LIN {X 0,Y 277.305,Z 271.444,A -85,B 0,C 180,E1 -17523.174,E2 -17523.174} C_VEL
LIN {X 0,Y 278.371,Z 274.382,A -85,B 0,C 180,E1 -17523.39,E2 -17523.39} C_VEL
LIN {X 0,Y 284.736,Z 287.887,A -85,B 0,C 180,E1 -17524.559,E2 -17524.559} C_VEL
LIN {X 0,Y 289.176,Z 296.03,A -85,B 0,C 180,E1 -17525.459,E2 -17525.459} C_VEL
LIN {X 0,Y 294.753,Z 304.53,A -85,B 0,C 180,E1 -17526.584,E2 -17526.584} C_VEL
LIN {X 0,Y 302.885,Z 314.906,A -85,B 0,C 180,E1 -17528.207,E2 -17528.207} C_VEL
LIN {X 0,Y 312.071,Z 325.664,A -85,B 0,C 180,E1 -17530.11,E2 -17530.11} C_VEL
LIN {X 0,Y 318.486,Z 332.585,A -85,B 0,C 180,E1 -17531.566,E2 -17531.566} C_VEL
LIN {X 0,Y 325.416,Z 339.712,A -85,B 0,C 180,E1 -17533.306,E2 -17533.306} C_VEL
LIN {X 0,Y 330.152,Z 344.132,A -85,B 0,C 180,E1 -17534.587,E2 -17534.587} C_VEL
LIN {X 0,Y 333.613,Z 347.56,A -85,B 0,C 180,E1 -17535.666,E2 -17535.666} C_VEL
LIN {X 0,Y 338.551,Z 351.983,A -85,B 0,C 180,E1 -17537.29,E2 -17537.29} C_VEL
LIN {X 0,Y 343.443,Z 356.189,A -85,B 0,C 180,E1 -17539.131,E2 -17539.131} C_VEL
LIN {X 0,Y 346.978,Z 358.993,A -85,B 0,C 180,E1 -17540.675,E2 -17540.675} C_VEL
LIN {X 0,Y 349.09,Z 361.115,A -85,B 0,C 180,E1 -17541.899,E2 -17541.899} C_VEL
LIN {X 0,Y 351.016,Z 362.827,A -85,B 0,C 180,E1 -17543.1,E2 -17543.1} C_VEL
LIN {X 0,Y 352.986,Z 364.25,A -85,B 0,C 180,E1 -17544.46,E2 -17544.46} C_VEL
LIN {X 0,Y 354.317,Z 364.994,A -85,B 0,C 180,E1 -17545.449,E2 -17545.449} C_VEL
LIN {X 0,Y 355.672,Z 365.56,A -85,B 0,C 180,E1 -17546.602,E2 -17546.602} C_VEL
LIN {X 0,Y 356.709,Z 365.873,A -85,B 0,C 180,E1 -17547.742,E2 -17547.742} C_VEL
LIN {X 0,Y 357.373,Z 366.011,A -85,B 0,C 180,E1 -17548.873,E2 -17548.873} C_VEL
LIN {X 0,Y 357.622,Z 366.036,A -85,B 0,C 180,E1 -17550,E2 -17550} C_VEL
LIN {X 0,Y 357.372,Z 366.013,A -85,B 0,C 180,E1 -17551.127,E2 -17551.127} C_VEL
LIN {X 0,Y 356.704,Z 365.874,A -85,B 0,C 180,E1 -17552.258,E2 -17552.258} C_VEL
LIN {X 0,Y 355.662,Z 365.563,A -85,B 0,C 180,E1 -17553.398,E2 -17553.398} C_VEL
LIN {X 0,Y 354.323,Z 364.997,A -85,B 0,C 180,E1 -17554.551,E2 -17554.551} C_VEL
LIN {X 0,Y 352.755,Z 364.109,A -85,B 0,C 180,E1 -17555.717,E2 -17555.717} C_VEL
LIN {X 0,Y 350.974,Z 362.834,A -85,B 0,C 180,E1 -17556.9,E2 -17556.9} C_VEL
LIN {X 0,Y 348.241,Z 360.258,A -85,B 0,C 180,E1 -17558.618,E2 -17558.618} C_VEL
LIN {X 0,Y 346.063,Z 358.167,A -85,B 0,C 180,E1 -17559.786,E2 -17559.786} C_VEL
LIN {X 0,Y 342.661,Z 355.63,A -85,B 0,C 180,E1 -17561.144,E2 -17561.144} C_VEL
LIN {X 0,Y 338.543,Z 351.93,A -85,B 0,C 180,E1 -17562.705,E2 -17562.705} C_VEL
LIN {X 0,Y 335.745,Z 349.331,A -85,B 0,C 180,E1 -17563.679,E2 -17563.679} C_VEL
LIN {X 0,Y 331.243,Z 345.273,A -85,B 0,C 180,E1 -17565.064,E2 -17565.064} C_VEL
LIN {X 0,Y 325.444,Z 339.675,A -85,B 0,C 180,E1 -17566.699,E2 -17566.699} C_VEL
LIN {X 0,Y 318.499,Z 332.541,A -85,B 0,C 180,E1 -17568.441,E2 -17568.441} C_VEL
LIN {X 0,Y 312.069,Z 325.652,A -85,B 0,C 180,E1 -17569.888,E2 -17569.888} C_VEL
LIN {X 0,Y 303.933,Z 316.233,A -85,B 0,C 180,E1 -17571.574,E2 -17571.574} C_VEL
LIN {X 0,Y 294.754,Z 304.541,A -85,B 0,C 180,E1 -17573.415,E2 -17573.415} C_VEL
LIN {X 0,Y 288.184,Z 294.427,A -85,B 0,C 180,E1 -17574.738,E2 -17574.738} C_VEL
LIN {X 0,Y 283.212,Z 284.587,A -85,B 0,C 180,E1 -17575.747,E2 -17575.747} C_VEL
LIN {X 0,Y 277.393,Z 272.078,A -85,B 0,C 180,E1 -17576.778,E2 -17576.778} C_VEL
LIN {X 0,Y 277.312,Z 271.443,A -85,B 0,C 180,E1 -17576.829,E2 -17576.829} C_VEL
LIN {X 0,Y 277.223,Z 271.454,A -85,B 0,C 180,E1 -17580.487,E2 -17580.487} C_VEL
LIN {X 0,Y 277.205,Z 271.457,A -85,B 0,C 180,E1 -17583.901,E2 -17583.901} C_VEL
LIN {X 0,Y 277.235,Z 271.451,A -85,B 0,C 180,E1 -17587.473,E2 -17587.473} C_VEL
LIN {X 0,Y 277.221,Z 271.451,A -85,B 0,C 180,E1 -17591.233,E2 -17591.233} C_VEL
LIN {X 0,Y 277.247,Z 271.448,A -85,B 0,C 180,E1 -17595.216,E2 -17595.216} C_VEL
LIN {X 0,Y 277.257,Z 271.449,A -85,B 0,C 180,E1 -17599.502,E2 -17599.502} C_VEL
LIN {X 0,Y 277.249,Z 271.448,A -85,B 0,C 180,E1 -17602.541,E2 -17602.541} C_VEL
LIN {X 0,Y 277.22,Z 271.451,A -85,B 0,C 180,E1 -17606.113,E2 -17606.113} C_VEL
LIN {X 0,Y 277.232,Z 271.453,A -85,B 0,C 180,E1 -17609.547,E2 -17609.547} C_VEL
LIN {X 0,Y 277.323,Z 271.439,A -85,B 0,C 180,E1 -17612.872,E2 -17612.872} C_VEL
LIN {X 0,Y 277.271,Z 271.444,A -85,B 0,C 180,E1 -17616.085,E2 -17616.085} C_VEL
LIN {X 0,Y 277.263,Z 271.443,A -85,B 0,C 180,E1 -17620.771,E2 -17620.771} C_VEL
LIN {X 0,Y 277.391,Z 271.43,A -85,B 0,C 180,E1 -17625.333,E2 -17625.333} C_VEL
LIN {X 0,Y 277.44,Z 271.421,A -85,B 0,C 180,E1 -17629.795,E2 -17629.795} C_VEL
LIN {X 0,Y 277.602,Z 271.406,A -85,B 0,C 180,E1 -17632.737,E2 -17632.737} C_VEL
LIN {X 0,Y 277.81,Z 271.365,A -85,B 0,C 180,E1 -17638.559,E2 -17638.559} C_VEL
LIN {X 0,Y 277.807,Z 271.377,A -85,B 0,C 180,E1 -17641.458,E2 -17641.458} C_VEL
LIN {X 0,Y 277.608,Z 271.404,A -85,B 0,C 180,E1 -17647.28,E2 -17647.28} C_VEL
LIN {X 0,Y 277.455,Z 271.425,A -85,B 0,C 180,E1 -17650.221,E2 -17650.221} C_VEL
LIN {X 0,Y 277.412,Z 271.431,A -85,B 0,C 180,E1 -17654.683,E2 -17654.683} C_VEL
LIN {X 0,Y 277.29,Z 271.443,A -85,B 0,C 180,E1 -17659.246,E2 -17659.246} C_VEL
LIN {X 0,Y 277.28,Z 271.448,A -85,B 0,C 180,E1 -17663.933,E2 -17663.933} C_VEL
LIN {X 0,Y 277.243,Z 271.447,A -85,B 0,C 180,E1 -17666.284,E2 -17666.284} C_VEL
LIN {X 0,Y 276.586,Z 271.534,A -85,B 0,C 180,E1 -17667.497,E2 -17667.497} C_VEL
LIN {X 0,Y 273.691,Z 271.893,A -85,B 0,C 180,E1 -17669.472,E2 -17669.472} C_VEL
LIN {X 0,Y 271.272,Z 272.333,A -85,B 0,C 180,E1 -17671.075,E2 -17671.075} C_VEL
LIN {X 0,Y 270.307,Z 272.789,A -85,B 0,C 180,E1 -17672.316,E2 -17672.316} C_VEL
LIN {X 0,Y 270.268,Z 272.974,A -85,B 0,C 180,E1 -17672.735,E2 -17672.735} C_VEL
LIN {X 0,Y 270.578,Z 275.102,A -85,B 0,C 180,E1 -17676.692,E2 -17676.692} C_VEL
LIN {X 0,Y 270.939,Z 277.348,A -85,B 0,C 180,E1 -17680.436,E2 -17680.436} C_VEL
LIN {X 0,Y 271.224,Z 279.969,A -85,B 0,C 180,E1 -17684.406,E2 -17684.406} C_VEL
LIN {X 0,Y 271.163,Z 282.305,A -85,B 0,C 180,E1 -17687.635,E2 -17687.635} C_VEL
LIN {X 0,Y 270.847,Z 285.048,A -85,B 0,C 180,E1 -17691.128,E2 -17691.128} C_VEL
LIN {X 0,Y 270.224,Z 288.327,A -85,B 0,C 180,E1 -17695.099,E2 -17695.099} C_VEL
LIN {X 0,Y 269.607,Z 292.063,A -85,B 0,C 180,E1 -17699.354,E2 -17699.354} C_VEL
LIN {X 0,Y 269.107,Z 295.022,A -85,B 0,C 180,E1 -17702.665,E2 -17702.665} C_VEL
LIN {X 0,Y 269.854,Z 298.046,A -85,B 0,C 180,E1 -17702.869,E2 -17702.869} C_VEL
LIN {X 0,Y 273.525,Z 311.599,A -85,B 0,C 180,E1 -17704.078,E2 -17704.078} C_VEL
LIN {X 0,Y 275.582,Z 321.927,A -85,B 0,C 180,E1 -17705.147,E2 -17705.147} C_VEL
LIN {X 0,Y 276.762,Z 330.171,A -85,B 0,C 180,E1 -17706.102,E2 -17706.102} C_VEL
LIN {X 0,Y 277.572,Z 339.948,A -85,B 0,C 180,E1 -17707.397,E2 -17707.397} C_VEL
LIN {X 0,Y 277.789,Z 344.628,A -85,B 0,C 180,E1 -17708.089,E2 -17708.089} C_VEL
LIN {X 0,Y 275.819,Z 355.141,A -85,B 0,C 180,E1 -17709.686,E2 -17709.686} C_VEL
LIN {X 0,Y 274.235,Z 363.639,A -85,B 0,C 180,E1 -17711.317,E2 -17711.317} C_VEL
LIN {X 0,Y 272.702,Z 371.465,A -85,B 0,C 180,E1 -17713.147,E2 -17713.147} C_VEL
LIN {X 0,Y 271.408,Z 378.004,A -85,B 0,C 180,E1 -17714.993,E2 -17714.993} C_VEL
LIN {X 0,Y 270.436,Z 382.504,A -85,B 0,C 180,E1 -17716.474,E2 -17716.474} C_VEL
LIN {X 0,Y 269.416,Z 387.997,A -85,B 0,C 180,E1 -17718.718,E2 -17718.718} C_VEL
LIN {X 0,Y 268.723,Z 392.325,A -85,B 0,C 180,E1 -17720.972,E2 -17720.972} C_VEL
LIN {X 0,Y 268.437,Z 394.694,A -85,B 0,C 180,E1 -17722.478,E2 -17722.478} C_VEL
LIN {X 0,Y 268.147,Z 397.425,A -85,B 0,C 180,E1 -17724.907,E2 -17724.907} C_VEL
LIN {X 0,Y 268.167,Z 398.948,A -85,B 0,C 180,E1 -17726.996,E2 -17726.996} C_VEL
LIN {X 0,Y 268.189,Z 399.539,A -85,B 0,C 180,E1 -17728.498,E2 -17728.498} C_VEL
LIN {X 0,Y 268.189,Z 399.539,A -85,B 0,C 180,E1 -17731.502,E2 -17731.502} C_VEL
LIN {X 0,Y 268.166,Z 398.948,A -85,B 0,C 180,E1 -17733.004,E2 -17733.004} C_VEL
LIN {X 0,Y 268.242,Z 396.496,A -85,B 0,C 180,E1 -17736.016,E2 -17736.016} C_VEL
LIN {X 0,Y 268.566,Z 393.543,A -85,B 0,C 180,E1 -17738.275,E2 -17738.275} C_VEL
LIN {X 0,Y 269.161,Z 389.552,A -85,B 0,C 180,E1 -17740.531,E2 -17740.531} C_VEL
LIN {X 0,Y 270.044,Z 384.42,A -85,B 0,C 180,E1 -17742.78,E2 -17742.78} C_VEL
LIN {X 0,Y 271.134,Z 379.159,A -85,B 0,C 180,E1 -17744.639,E2 -17744.639} C_VEL
LIN {X 0,Y 272.4,Z 372.841,A -85,B 0,C 180,E1 -17746.487,E2 -17746.487} C_VEL
LIN {X 0,Y 273.641,Z 366.891,A -85,B 0,C 180,E1 -17747.95,E2 -17747.95} C_VEL
LIN {X 0,Y 274.86,Z 359.961,A -85,B 0,C 180,E1 -17749.414,E2 -17749.414} C_VEL
LIN {X 0,Y 276.443,Z 351.784,A -85,B 0,C 180,E1 -17750.849,E2 -17750.849} C_VEL
LIN {X 0,Y 277.754,Z 344.627,A -85,B 0,C 180,E1 -17751.914,E2 -17751.914} C_VEL
LIN {X 0,Y 277.272,Z 335.68,A -85,B 0,C 180,E1 -17753.188,E2 -17753.188} C_VEL
LIN {X 0,Y 276.143,Z 325.328,A -85,B 0,C 180,E1 -17754.463,E2 -17754.463} C_VEL
LIN {X 0,Y 274.461,Z 315.993,A -85,B 0,C 180,E1 -17755.483,E2 -17755.483} C_VEL
LIN {X 0,Y 271.884,Z 305.118,A -85,B 0,C 180,E1 -17756.518,E2 -17756.518} C_VEL
LIN {X 0,Y 269.171,Z 295.65,A -85,B 0,C 180,E1 -17757.299,E2 -17757.299} C_VEL
LIN {X 0,Y 269.089,Z 295.013,A -85,B 0,C 180,E1 -17757.365,E2 -17757.365} C_VEL
LIN {X 0,Y 269.661,Z 291.299,A -85,B 0,C 180,E1 -17761.415,E2 -17761.415} C_VEL
LIN {X 0,Y 270.24,Z 288.287,A -85,B 0,C 180,E1 -17764.899,E2 -17764.899} C_VEL
LIN {X 0,Y 270.846,Z 285.017,A -85,B 0,C 180,E1 -17768.872,E2 -17768.872} C_VEL
LIN {X 0,Y 271.157,Z 282.304,A -85,B 0,C 180,E1 -17772.366,E2 -17772.366} C_VEL
LIN {X 0,Y 271.224,Z 279.957,A -85,B 0,C 180,E1 -17775.594,E2 -17775.594} C_VEL
LIN {X 0,Y 270.939,Z 277.339,A -85,B 0,C 180,E1 -17779.564,E2 -17779.564} C_VEL
LIN {X 0,Y 270.556,Z 274.906,A -85,B 0,C 180,E1 -17783.633,E2 -17783.633} C_VEL
LIN {X 0,Y 270.315,Z 273.144,A -85,B 0,C 180,E1 -17786.9,E2 -17786.9} C_VEL
LIN {X 0,Y 270.196,Z 272.332,A -85,B 0,C 180,E1 -17789.13,E2 -17789.13} C_VEL
LIN {X 0,Y 270.209,Z 272.329,A -85,B 0,C 180,E1 -17792.166,E2 -17792.166} C_VEL
LIN {X 0,Y 270.226,Z 272.327,A -85,B 0,C 180,E1 -17795.54,E2 -17795.54} C_VEL
LIN {X 0,Y 270.23,Z 272.325,A -85,B 0,C 180,E1 -17800.231,E2 -17800.231} C_VEL
LIN {X 0,Y 270.371,Z 272.305,A -85,B 0,C 180,E1 -17804.926,E2 -17804.926} C_VEL
LIN {X 0,Y 270.407,Z 272.304,A -85,B 0,C 180,E1 -17809.509,E2 -17809.509} C_VEL
LIN {X 0,Y 270.568,Z 272.28,A -85,B 0,C 180,E1 -17812.529,E2 -17812.529} C_VEL
LIN {X 0,Y 270.771,Z 272.253,A -85,B 0,C 180,E1 -17818.504,E2 -17818.504} C_VEL
LIN {X 0,Y 270.776,Z 272.239,A -85,B 0,C 180,E1 -17821.479,E2 -17821.479} C_VEL
LIN {X 0,Y 270.562,Z 272.282,A -85,B 0,C 180,E1 -17827.453,E2 -17827.453} C_VEL
LIN {X 0,Y 270.392,Z 272.3,A -85,B 0,C 180,E1 -17830.473,E2 -17830.473} C_VEL
LIN {X 0,Y 270.35,Z 272.307,A -85,B 0,C 180,E1 -17835.058,E2 -17835.058} C_VEL
LIN {X 0,Y 270.202,Z 272.321,A -85,B 0,C 180,E1 -17839.753,E2 -17839.753} C_VEL
LIN {X 0,Y 270.212,Z 272.324,A -85,B 0,C 180,E1 -17844.58,E2 -17844.58} C_VEL
LIN {X 0,Y 270.217,Z 272.324,A -85,B 0,C 180,E1 -17847.903,E2 -17847.903} C_VEL
LIN {X 0,Y 270.143,Z 272.333,A -85,B 0,C 180,E1 -17851.341,E2 -17851.341} C_VEL
LIN {X 0,Y 270.181,Z 272.329,A -85,B 0,C 180,E1 -17854.895,E2 -17854.895} C_VEL
LIN {X 0,Y 270.187,Z 272.329,A -85,B 0,C 180,E1 -17858.709,E2 -17858.709} C_VEL
LIN {X 0,Y 270.191,Z 272.329,A -85,B 0,C 180,E1 -17862.539,E2 -17862.539} C_VEL
LIN {X 0,Y 270.19,Z 272.327,A -85,B 0,C 180,E1 -17866.729,E2 -17866.729} C_VEL
LIN {X 0,Y 270.202,Z 272.326,A -85,B 0,C 180,E1 -17869.441,E2 -17869.441} C_VEL
LIN {X 0,Y 270.207,Z 272.328,A -85,B 0,C 180,E1 -17873.716,E2 -17873.716} C_VEL
LIN {X 0,Y 270.155,Z 272.333,A -85,B 0,C 180,E1 -17876.887,E2 -17876.887} C_VEL
LIN {X 0,Y 270.178,Z 272.331,A -85,B 0,C 180,E1 -17880.381,E2 -17880.381} C_VEL
LIN {X 0,Y 270.246,Z 272.322,A -85,B 0,C 180,E1 -17882.435,E2 -17882.435} C_VEL
LIN {X 0,Y 271.193,Z 275.036,A -85,B 0,C 180,E1 -17882.64,E2 -17882.64} C_VEL
LIN {X 0,Y 277.258,Z 287.788,A -85,B 0,C 180,E1 -17883.803,E2 -17883.803} C_VEL
LIN {X 0,Y 281.67,Z 296.983,A -85,B 0,C 180,E1 -17884.809,E2 -17884.809} C_VEL
LIN {X 0,Y 287.233,Z 305.985,A -85,B 0,C 180,E1 -17886.041,E2 -17886.041} C_VEL
LIN {X 0,Y 294.832,Z 316.369,A -85,B 0,C 180,E1 -17887.711,E2 -17887.711} C_VEL
LIN {X 0,Y 304.031,Z 327.199,A -85,B 0,C 180,E1 -17889.712,E2 -17889.712} C_VEL
LIN {X 0,Y 312.544,Z 336.483,A -85,B 0,C 180,E1 -17891.651,E2 -17891.651} C_VEL
LIN {X 0,Y 318.048,Z 342.107,A -85,B 0,C 180,E1 -17893.005,E2 -17893.005} C_VEL
LIN {X 0,Y 324.198,Z 348.021,A -85,B 0,C 180,E1 -17894.649,E2 -17894.649} C_VEL
LIN {X 0,Y 328.692,Z 352.374,A -85,B 0,C 180,E1 -17896.035,E2 -17896.035} C_VEL
LIN {X 0,Y 333.966,Z 357.233,A -85,B 0,C 180,E1 -17897.852,E2 -17897.852} C_VEL
LIN {X 0,Y 338.688,Z 361.032,A -85,B 0,C 180,E1 -17899.64,E2 -17899.64} C_VEL
LIN {X 0,Y 341.529,Z 363.397,A -85,B 0,C 180,E1 -17900.955,E2 -17900.955} C_VEL
LIN {X 0,Y 344.893,Z 366.614,A -85,B 0,C 180,E1 -17902.977,E2 -17902.977} C_VEL
LIN {X 0,Y 346.673,Z 368.004,A -85,B 0,C 180,E1 -17904.182,E2 -17904.182} C_VEL
LIN {X 0,Y 348.314,Z 368.949,A -85,B 0,C 180,E1 -17905.371,E2 -17905.371} C_VEL
LIN {X 0,Y 349.715,Z 369.542,A -85,B 0,C 180,E1 -17906.544,E2 -17906.544} C_VEL
LIN {X 0,Y 350.797,Z 369.895,A -85,B 0,C 180,E1 -17907.704,E2 -17907.704} C_VEL
LIN {X 0,Y 351.516,Z 370.064,A -85,B 0,C 180,E1 -17908.854,E2 -17908.854} C_VEL
LIN {X 0,Y 351.802,Z 370.093,A -85,B 0,C 180,E1 -17910,E2 -17910} C_VEL
LIN {X 0,Y 351.428,Z 370.042,A -85,B 0,C 180,E1 -17911.304,E2 -17911.304} C_VEL
LIN {X 0,Y 350.795,Z 369.894,A -85,B 0,C 180,E1 -17912.296,E2 -17912.296} C_VEL
LIN {X 0,Y 349.687,Z 369.557,A -85,B 0,C 180,E1 -17913.457,E2 -17913.457} C_VEL
LIN {X 0,Y 348.32,Z 368.954,A -85,B 0,C 180,E1 -17914.629,E2 -17914.629} C_VEL
LIN {X 0,Y 346.271,Z 367.704,A -85,B 0,C 180,E1 -17916.102,E2 -17916.102} C_VEL
LIN {X 0,Y 342.923,Z 364.794,A -85,B 0,C 180,E1 -17918.248,E2 -17918.248} C_VEL
LIN {X 0,Y 340.682,Z 362.566,A -85,B 0,C 180,E1 -17919.499,E2 -17919.499} C_VEL
LIN {X 0,Y 336.609,Z 359.463,A -85,B 0,C 180,E1 -17921.151,E2 -17921.151} C_VEL
LIN {X 0,Y 333.301,Z 356.536,A -85,B 0,C 180,E1 -17922.404,E2 -17922.404} C_VEL
LIN {X 0,Y 328.614,Z 352.291,A -85,B 0,C 180,E1 -17923.982,E2 -17923.982} C_VEL
LIN {X 0,Y 323.151,Z 347.015,A -85,B 0,C 180,E1 -17925.649,E2 -17925.649} C_VEL
LIN {X 0,Y 316.588,Z 340.622,A -85,B 0,C 180,E1 -17927.374,E2 -17927.374} C_VEL
LIN {X 0,Y 310.388,Z 334.142,A -85,B 0,C 180,E1 -17928.866,E2 -17928.866} C_VEL
LIN {X 0,Y 300.983,Z 323.659,A -85,B 0,C 180,E1 -17930.963,E2 -17930.963} C_VEL
LIN {X 0,Y 292.248,Z 312.969,A -85,B 0,C 180,E1 -17932.863,E2 -17932.863} C_VEL
LIN {X 0,Y 285.391,Z 303.244,A -85,B 0,C 180,E1 -17934.362,E2 -17934.362} C_VEL
LIN {X 0,Y 279.96,Z 293.672,A -85,B 0,C 180,E1 -17935.584,E2 -17935.584} C_VEL
LIN {X 0,Y 273.934,Z 280.583,A -85,B 0,C 180,E1 -17936.873,E2 -17936.873} C_VEL
LIN {X 0,Y 270.418,Z 273.239,A -85,B 0,C 180,E1 -17937.498,E2 -17937.498} C_VEL
LIN {X 0,Y 270.232,Z 272.324,A -85,B 0,C 180,E1 -17937.598,E2 -17937.598} C_VEL
LIN {X 0,Y 270.135,Z 272.335,A -85,B 0,C 180,E1 -17941.354,E2 -17941.354} C_VEL
LIN {X 0,Y 270.166,Z 272.331,A -85,B 0,C 180,E1 -17944.91,E2 -17944.91} C_VEL
LIN {X 0,Y 270.178,Z 272.329,A -85,B 0,C 180,E1 -17948.723,E2 -17948.723} C_VEL
LIN {X 0,Y 270.187,Z 272.328,A -85,B 0,C 180,E1 -17952.554,E2 -17952.554} C_VEL
LIN {X 0,Y 270.192,Z 272.327,A -85,B 0,C 180,E1 -17956.743,E2 -17956.743} C_VEL
LIN {X 0,Y 270.209,Z 272.327,A -85,B 0,C 180,E1 -17959.455,E2 -17959.455} C_VEL
LIN {X 0,Y 270.221,Z 272.326,A -85,B 0,C 180,E1 -17963.73,E2 -17963.73} C_VEL
LIN {X 0,Y 270.17,Z 272.329,A -85,B 0,C 180,E1 -17966.901,E2 -17966.901} C_VEL
LIN {X 0,Y 270.162,Z 272.331,A -85,B 0,C 180,E1 -17970.391,E2 -17970.391} C_VEL
LIN {X 0,Y 270.229,Z 272.322,A -85,B 0,C 180,E1 -17973.772,E2 -17973.772} C_VEL
LIN {X 0,Y 270.182,Z 272.329,A -85,B 0,C 180,E1 -17977.045,E2 -17977.045} C_VEL
LIN {X 0,Y 270.202,Z 272.321,A -85,B 0,C 180,E1 -17980.247,E2 -17980.247} C_VEL
LIN {X 0,Y 270.35,Z 272.307,A -85,B 0,C 180,E1 -17984.942,E2 -17984.942} C_VEL
LIN {X 0,Y 270.392,Z 272.3,A -85,B 0,C 180,E1 -17989.527,E2 -17989.527} C_VEL
LIN {X 0,Y 270.562,Z 272.282,A -85,B 0,C 180,E1 -17992.547,E2 -17992.547} C_VEL
LIN {X 0,Y 270.776,Z 272.239,A -85,B 0,C 180,E1 -17998.521,E2 -17998.521} C_VEL
LIN {X 0,Y 270.771,Z 272.253,A -85,B 0,C 180,E1 -18001.496,E2 -18001.496} C_VEL
LIN {X 0,Y 270.568,Z 272.28,A -85,B 0,C 180,E1 -18007.471,E2 -18007.471} C_VEL
LIN {X 0,Y 270.407,Z 272.305,A -85,B 0,C 180,E1 -18010.491,E2 -18010.491} C_VEL
LIN {X 0,Y 270.371,Z 272.306,A -85,B 0,C 180,E1 -18015.074,E2 -18015.074} C_VEL
LIN {X 0,Y 270.229,Z 272.324,A -85,B 0,C 180,E1 -18019.769,E2 -18019.769} C_VEL
LIN {X 0,Y 270.207,Z 272.328,A -85,B 0,C 180,E1 -18024.6,E2 -18024.6} C_VEL
LIN {X 0,Y 270.206,Z 272.328,A -85,B 0,C 180,E1 -18027.924,E2 -18027.924} C_VEL
LIN {X 0,Y 270.187,Z 272.334,A -85,B 0,C 180,E1 -18031.356,E2 -18031.356} C_VEL
LIN {X 0,Y 270.268,Z 272.974,A -85,B 0,C 180,E1 -18032.735,E2 -18032.735} C_VEL
LIN {X 0,Y 269.724,Z 273.708,A -85,B 0,C 180,E1 -18033.973,E2 -18033.973} C_VEL
LIN {X 0,Y 267.004,Z 275.236,A -85,B 0,C 180,E1 -18035.983,E2 -18035.983} C_VEL
LIN {X 0,Y 264.697,Z 276.523,A -85,B 0,C 180,E1 -18037.616,E2 -18037.616} C_VEL
LIN {X 0,Y 263.792,Z 277.402,A -85,B 0,C 180,E1 -18038.882,E2 -18038.882} C_VEL
LIN {X 0,Y 263.768,Z 277.665,A -85,B 0,C 180,E1 -18039.311,E2 -18039.311} C_VEL
LIN {X 0,Y 263.995,Z 279.198,A -85,B 0,C 180,E1 -18041.807,E2 -18041.807} C_VEL
LIN {X 0,Y 264.161,Z 280.692,A -85,B 0,C 180,E1 -18044.084,E2 -18044.084} C_VEL
LIN {X 0,Y 264.182,Z 282.173,A -85,B 0,C 180,E1 -18046.239,E2 -18046.239} C_VEL
LIN {X 0,Y 264.084,Z 283.666,A -85,B 0,C 180,E1 -18048.294,E2 -18048.294} C_VEL
LIN {X 0,Y 263.6,Z 286.669,A -85,B 0,C 180,E1 -18052.179,E2 -18052.179} C_VEL
LIN {X 0,Y 263.009,Z 289.753,A -85,B 0,C 180,E1 -18055.942,E2 -18055.942} C_VEL
LIN {X 0,Y 262.512,Z 292.712,A -85,B 0,C 180,E1 -18059.426,E2 -18059.426} C_VEL
LIN {X 0,Y 262.102,Z 294.933,A -85,B 0,C 180,E1 -18061.88,E2 -18061.88} C_VEL
LIN {X 0,Y 263.003,Z 298.178,A -85,B 0,C 180,E1 -18062.116,E2 -18062.116} C_VEL
LIN {X 0,Y 266.675,Z 311.678,A -85,B 0,C 180,E1 -18063.384,E2 -18063.384} C_VEL
LIN {X 0,Y 268.682,Z 321.718,A -85,B 0,C 180,E1 -18064.464,E2 -18064.464} C_VEL
LIN {X 0,Y 270.078,Z 331.206,A -85,B 0,C 180,E1 -18065.626,E2 -18065.626} C_VEL
LIN {X 0,Y 270.79,Z 339.979,A -85,B 0,C 180,E1 -18066.833,E2 -18066.833} C_VEL
LIN {X 0,Y 270.977,Z 345.785,A -85,B 0,C 180,E1 -18067.71,E2 -18067.71} C_VEL
LIN {X 0,Y 268.939,Z 355.928,A -85,B 0,C 180,E1 -18069.343,E2 -18069.343} C_VEL
LIN {X 0,Y 267.111,Z 365.231,A -85,B 0,C 180,E1 -18071.238,E2 -18071.238} C_VEL
LIN {X 0,Y 265.889,Z 371.318,A -85,B 0,C 180,E1 -18072.715,E2 -18072.715} C_VEL
LIN {X 0,Y 264.53,Z 377.808,A -85,B 0,C 180,E1 -18074.593,E2 -18074.593} C_VEL
LIN {X 0,Y 263.527,Z 382.309,A -85,B 0,C 180,E1 -18076.113,E2 -18076.113} C_VEL
LIN {X 0,Y 262.425,Z 387.802,A -85,B 0,C 180,E1 -18078.413,E2 -18078.413} C_VEL
LIN {X 0,Y 261.702,Z 392.13,A -85,B 0,C 180,E1 -18080.728,E2 -18080.728} C_VEL
LIN {X 0,Y 261.372,Z 394.499,A -85,B 0,C 180,E1 -18082.274,E2 -18082.274} C_VEL
LIN {X 0,Y 261.046,Z 397.423,A -85,B 0,C 180,E1 -18085.02,E2 -18085.02} C_VEL
LIN {X 0,Y 261.062,Z 398.753,A -85,B 0,C 180,E1 -18086.914,E2 -18086.914} C_VEL
LIN {X 0,Y 261.095,Z 399.345,A -85,B 0,C 180,E1 -18088.458,E2 -18088.458} C_VEL
LIN {X 0,Y 261.095,Z 399.345,A -85,B 0,C 180,E1 -18091.542,E2 -18091.542} C_VEL
LIN {X 0,Y 261.061,Z 398.753,A -85,B 0,C 180,E1 -18093.086,E2 -18093.086} C_VEL
LIN {X 0,Y 261.17,Z 396.301,A -85,B 0,C 180,E1 -18096.179,E2 -18096.179} C_VEL
LIN {X 0,Y 261.528,Z 393.348,A -85,B 0,C 180,E1 -18098.499,E2 -18098.499} C_VEL
LIN {X 0,Y 262.137,Z 389.356,A -85,B 0,C 180,E1 -18100.817,E2 -18100.817} C_VEL
LIN {X 0,Y 263.103,Z 384.224,A -85,B 0,C 180,E1 -18103.123,E2 -18103.123} C_VEL
LIN {X 0,Y 264.253,Z 378.963,A -85,B 0,C 180,E1 -18105.029,E2 -18105.029} C_VEL
LIN {X 0,Y 265.586,Z 372.646,A -85,B 0,C 180,E1 -18106.922,E2 -18106.922} C_VEL
LIN {X 0,Y 266.839,Z 366.695,A -85,B 0,C 180,E1 -18108.424,E2 -18108.424} C_VEL
LIN {X 0,Y 268.137,Z 359.766,A -85,B 0,C 180,E1 -18109.921,E2 -18109.921} C_VEL
LIN {X 0,Y 269.814,Z 351.589,A -85,B 0,C 180,E1 -18111.386,E2 -18111.386} C_VEL
LIN {X 0,Y 270.986,Z 344.427,A -85,B 0,C 180,E1 -18112.49,E2 -18112.49} C_VEL
LIN {X 0,Y 270.41,Z 335.182,A -85,B 0,C 180,E1 -18113.849,E2 -18113.849} C_VEL
LIN {X 0,Y 269.366,Z 325.614,A -85,B 0,C 180,E1 -18115.071,E2 -18115.071} C_VEL
LIN {X 0,Y 267.439,Z 315.176,A -85,B 0,C 180,E1 -18116.252,E2 -18116.252} C_VEL
LIN {X 0,Y 265.009,Z 305.206,A -85,B 0,C 180,E1 -18117.244,E2 -18117.244} C_VEL
LIN {X 0,Y 262.166,Z 295.677,A -85,B 0,C 180,E1 -18118.082,E2 -18118.082} C_VEL
LIN {X 0,Y 262.101,Z 294.855,A -85,B 0,C 180,E1 -18118.14,E2 -18118.14} C_VEL
LIN {X 0,Y 262.547,Z 292.237,A -85,B 0,C 180,E1 -18121.052,E2 -18121.052} C_VEL
LIN {X 0,Y 263.02,Z 289.659,A -85,B 0,C 180,E1 -18124.133,E2 -18124.133} C_VEL
LIN {X 0,Y 263.6,Z 286.643,A -85,B 0,C 180,E1 -18127.821,E2 -18127.821} C_VEL
LIN {X 0,Y 264.084,Z 283.661,A -85,B 0,C 180,E1 -18131.706,E2 -18131.706} C_VEL
LIN {X 0,Y 264.186,Z 281.942,A -85,B 0,C 180,E1 -18134.079,E2 -18134.079} C_VEL
LIN {X 0,Y 264.144,Z 280.466,A -85,B 0,C 180,E1 -18136.22,E2 -18136.22} C_VEL
LIN {X 0,Y 264.015,Z 279.143,A -85,B 0,C 180,E1 -18138.271,E2 -18138.271} C_VEL
LIN {X 0,Y 263.644,Z 276.792,A -85,B 0,C 180,E1 -18142.176,E2 -18142.176} C_VEL
LIN {X 0,Y 263.361,Z 274.743,A -85,B 0,C 180,E1 -18145.908,E2 -18145.908} C_VEL
LIN {X 0,Y 263.161,Z 273.351,A -85,B 0,C 180,E1 -18148.713,E2 -18148.713} C_VEL
LIN {X 0,Y 263.137,Z 273.207,A -85,B 0,C 180,E1 -18152.988,E2 -18152.988} C_VEL
LIN {X 0,Y 263.145,Z 273.208,A -85,B 0,C 180,E1 -18156.375,E2 -18156.375} C_VEL
LIN {X 0,Y 263.215,Z 273.201,A -85,B 0,C 180,E1 -18159.681,E2 -18159.681} C_VEL
LIN {X 0,Y 263.314,Z 273.184,A -85,B 0,C 180,E1 -18164.511,E2 -18164.511} C_VEL
LIN {X 0,Y 263.346,Z 273.182,A -85,B 0,C 180,E1 -18169.225,E2 -18169.225} C_VEL
LIN {X 0,Y 263.531,Z 273.157,A -85,B 0,C 180,E1 -18172.329,E2 -18172.329} C_VEL
LIN {X 0,Y 263.734,Z 273.129,A -85,B 0,C 180,E1 -18178.464,E2 -18178.464} C_VEL
LIN {X 0,Y 263.74,Z 273.114,A -85,B 0,C 180,E1 -18181.518,E2 -18181.518} C_VEL
LIN {X 0,Y 263.523,Z 273.158,A -85,B 0,C 180,E1 -18187.654,E2 -18187.654} C_VEL
LIN {X 0,Y 263.331,Z 273.181,A -85,B 0,C 180,E1 -18190.758,E2 -18190.758} C_VEL
LIN {X 0,Y 263.292,Z 273.186,A -85,B 0,C 180,E1 -18195.471,E2 -18195.471} C_VEL
LIN {X 0,Y 263.187,Z 273.196,A -85,B 0,C 180,E1 -18200.302,E2 -18200.302} C_VEL
LIN {X 0,Y 263.165,Z 273.2,A -85,B 0,C 180,E1 -18205.284,E2 -18205.284} C_VEL
LIN {X 0,Y 263.126,Z 273.21,A -85,B 0,C 180,E1 -18208.724,E2 -18208.724} C_VEL
LIN {X 0,Y 263.097,Z 273.214,A -85,B 0,C 180,E1 -18212.28,E2 -18212.28} C_VEL
LIN {X 0,Y 263.154,Z 273.205,A -85,B 0,C 180,E1 -18215.97,E2 -18215.97} C_VEL
LIN {X 0,Y 263.123,Z 273.21,A -85,B 0,C 180,E1 -18219.855,E2 -18219.855} C_VEL
LIN {X 0,Y 263.151,Z 273.207,A -85,B 0,C 180,E1 -18223.962,E2 -18223.962} C_VEL
LIN {X 0,Y 263.128,Z 273.211,A -85,B 0,C 180,E1 -18228.109,E2 -18228.109} C_VEL
LIN {X 0,Y 263.142,Z 273.209,A -85,B 0,C 180,E1 -18232.101,E2 -18232.101} C_VEL
LIN {X 0,Y 263.137,Z 273.209,A -85,B 0,C 180,E1 -18235.884,E2 -18235.884} C_VEL
LIN {X 0,Y 263.101,Z 273.213,A -85,B 0,C 180,E1 -18239.501,E2 -18239.501} C_VEL
LIN {X 0,Y 263.174,Z 273.347,A -85,B 0,C 180,E1 -18241.674,E2 -18241.674} C_VEL
LIN {X 0,Y 264.168,Z 276.039,A -85,B 0,C 180,E1 -18241.873,E2 -18241.873} C_VEL
LIN {X 0,Y 270.002,Z 287.895,A -85,B 0,C 180,E1 -18243.037,E2 -18243.037} C_VEL
LIN {X 0,Y 274.745,Z 298.532,A -85,B 0,C 180,E1 -18244.224,E2 -18244.224} C_VEL
LIN {X 0,Y 279.966,Z 307.797,A -85,B 0,C 180,E1 -18245.523,E2 -18245.523} C_VEL
LIN {X 0,Y 286.211,Z 316.753,A -85,B 0,C 180,E1 -18247.016,E2 -18247.016} C_VEL
LIN {X 0,Y 294.917,Z 327.456,A -85,B 0,C 180,E1 -18249.056,E2 -18249.056} C_VEL
LIN {X 0,Y 304.221,Z 337.698,A -85,B 0,C 180,E1 -18251.257,E2 -18251.257} C_VEL
LIN {X 0,Y 311.996,Z 345.716,A -85,B 0,C 180,E1 -18253.166,E2 -18253.166} C_VEL
LIN {X 0,Y 318.525,Z 352.006,A -85,B 0,C 180,E1 -18254.938,E2 -18254.938} C_VEL
LIN {X 0,Y 322.402,Z 355.804,A -85,B 0,C 180,E1 -18256.126,E2 -18256.126} C_VEL
LIN {X 0,Y 326.785,Z 359.743,A -85,B 0,C 180,E1 -18257.581,E2 -18257.581} C_VEL
LIN {X 0,Y 330.501,Z 363.053,A -85,B 0,C 180,E1 -18258.967,E2 -18258.967} C_VEL
LIN {X 0,Y 334.685,Z 366.228,A -85,B 0,C 180,E1 -18260.666,E2 -18260.666} C_VEL
LIN {X 0,Y 338.411,Z 369.858,A -85,B 0,C 180,E1 -18262.842,E2 -18262.842} C_VEL
LIN {X 0,Y 340.265,Z 371.35,A -85,B 0,C 180,E1 -18264.073,E2 -18264.073} C_VEL
LIN {X 0,Y 341.945,Z 372.35,A -85,B 0,C 180,E1 -18265.284,E2 -18265.284} C_VEL
LIN {X 0,Y 343.406,Z 373.025,A -85,B 0,C 180,E1 -18266.48,E2 -18266.48} C_VEL
LIN {X 0,Y 344.592,Z 373.444,A -85,B 0,C 180,E1 -18267.679,E2 -18267.679} C_VEL
LIN {X 0,Y 345.365,Z 373.648,A -85,B 0,C 180,E1 -18268.834,E2 -18268.834} C_VEL
LIN {X 0,Y 345.687,Z 373.691,A -85,B 0,C 180,E1 -18270,E2 -18270} C_VEL
LIN {X 0,Y 345.385,Z 373.638,A -85,B 0,C 180,E1 -18271.166,E2 -18271.166} C_VEL
LIN {X 0,Y 344.56,Z 373.447,A -85,B 0,C 180,E1 -18272.338,E2 -18272.338} C_VEL
LIN {X 0,Y 343.372,Z 373.043,A -85,B 0,C 180,E1 -18273.52,E2 -18273.52} C_VEL
LIN {X 0,Y 341.954,Z 372.356,A -85,B 0,C 180,E1 -18274.715,E2 -18274.715} C_VEL
LIN {X 0,Y 339.444,Z 370.751,A -85,B 0,C 180,E1 -18276.47,E2 -18276.47} C_VEL
LIN {X 0,Y 336.389,Z 367.91,A -85,B 0,C 180,E1 -18278.409,E2 -18278.409} C_VEL
LIN {X 0,Y 333.836,Z 365.618,A -85,B 0,C 180,E1 -18279.696,E2 -18279.696} C_VEL
LIN {X 0,Y 328.688,Z 361.483,A -85,B 0,C 180,E1 -18281.719,E2 -18281.719} C_VEL
LIN {X 0,Y 323.601,Z 356.804,A -85,B 0,C 180,E1 -18283.51,E2 -18283.51} C_VEL
LIN {X 0,Y 318.506,Z 352.015,A -85,B 0,C 180,E1 -18285.07,E2 -18285.07} C_VEL
LIN {X 0,Y 311.999,Z 345.711,A -85,B 0,C 180,E1 -18286.836,E2 -18286.836} C_VEL
LIN {X 0,Y 303.534,Z 336.933,A -85,B 0,C 180,E1 -18288.914,E2 -18288.914} C_VEL
LIN {X 0,Y 292.987,Z 325.208,A -85,B 0,C 180,E1 -18291.392,E2 -18291.392} C_VEL
LIN {X 0,Y 284.418,Z 314.381,A -85,B 0,C 180,E1 -18293.408,E2 -18293.408} C_VEL
LIN {X 0,Y 278.042,Z 304.538,A -85,B 0,C 180,E1 -18294.961,E2 -18294.961} C_VEL
LIN {X 0,Y 273.081,Z 295.141,A -85,B 0,C 180,E1 -18296.19,E2 -18296.19} C_VEL
LIN {X 0,Y 267.373,Z 282.256,A -85,B 0,C 180,E1 -18297.529,E2 -18297.529} C_VEL
LIN {X 0,Y 263.315,Z 274.054,A -85,B 0,C 180,E1 -18298.288,E2 -18298.288} C_VEL
LIN {X 0,Y 263.15,Z 273.208,A -85,B 0,C 180,E1 -18298.367,E2 -18298.367} C_VEL
LIN {X 0,Y 263.084,Z 273.216,A -85,B 0,C 180,E1 -18302.294,E2 -18302.294} C_VEL
LIN {X 0,Y 263.14,Z 273.209,A -85,B 0,C 180,E1 -18305.985,E2 -18305.985} C_VEL
LIN {X 0,Y 263.117,Z 273.212,A -85,B 0,C 180,E1 -18309.869,E2 -18309.869} C_VEL
LIN {X 0,Y 263.15,Z 273.207,A -85,B 0,C 180,E1 -18313.977,E2 -18313.977} C_VEL
LIN {X 0,Y 263.133,Z 273.209,A -85,B 0,C 180,E1 -18318.124,E2 -18318.124} C_VEL
LIN {X 0,Y 263.153,Z 273.206,A -85,B 0,C 180,E1 -18322.116,E2 -18322.116} C_VEL
LIN {X 0,Y 263.152,Z 273.205,A -85,B 0,C 180,E1 -18325.899,E2 -18325.899} C_VEL
LIN {X 0,Y 263.098,Z 273.213,A -85,B 0,C 180,E1 -18329.513,E2 -18329.513} C_VEL
LIN {X 0,Y 263.161,Z 273.204,A -85,B 0,C 180,E1 -18333.011,E2 -18333.011} C_VEL
LIN {X 0,Y 263.128,Z 273.206,A -85,B 0,C 180,E1 -18336.393,E2 -18336.393} C_VEL
LIN {X 0,Y 263.187,Z 273.196,A -85,B 0,C 180,E1 -18339.698,E2 -18339.698} C_VEL
LIN {X 0,Y 263.292,Z 273.186,A -85,B 0,C 180,E1 -18344.529,E2 -18344.529} C_VEL
LIN {X 0,Y 263.331,Z 273.181,A -85,B 0,C 180,E1 -18349.242,E2 -18349.242} C_VEL
LIN {X 0,Y 263.523,Z 273.158,A -85,B 0,C 180,E1 -18352.346,E2 -18352.346} C_VEL
LIN {X 0,Y 263.74,Z 273.114,A -85,B 0,C 180,E1 -18358.482,E2 -18358.482} C_VEL
LIN {X 0,Y 263.734,Z 273.129,A -85,B 0,C 180,E1 -18361.536,E2 -18361.536} C_VEL
LIN {X 0,Y 263.531,Z 273.157,A -85,B 0,C 180,E1 -18367.671,E2 -18367.671} C_VEL
LIN {X 0,Y 263.346,Z 273.183,A -85,B 0,C 180,E1 -18370.775,E2 -18370.775} C_VEL
LIN {X 0,Y 263.314,Z 273.185,A -85,B 0,C 180,E1 -18375.489,E2 -18375.489} C_VEL
LIN {X 0,Y 263.215,Z 273.2,A -85,B 0,C 180,E1 -18380.319,E2 -18380.319} C_VEL
LIN {X 0,Y 263.145,Z 273.208,A -85,B 0,C 180,E1 -18385.306,E2 -18385.306} C_VEL
LIN {X 0,Y 263.14,Z 273.208,A -85,B 0,C 180,E1 -18388.743,E2 -18388.743} C_VEL
LIN {X 0,Y 263.161,Z 273.35,A -85,B 0,C 180,E1 -18391.287,E2 -18391.287} C_VEL
LIN {X 0,Y 263.359,Z 274.803,A -85,B 0,C 180,E1 -18394.183,E2 -18394.183} C_VEL
LIN {X 0,Y 263.644,Z 276.792,A -85,B 0,C 180,E1 -18397.824,E2 -18397.824} C_VEL
LIN {X 0,Y 263.768,Z 277.665,A -85,B 0,C 180,E1 -18399.311,E2 -18399.311} C_VEL
LIN {X 0,Y 263.263,Z 278.518,A -85,B 0,C 180,E1 -18400.574,E2 -18400.574} C_VEL
LIN {X 0,Y 260.575,Z 280.205,A -85,B 0,C 180,E1 -18402.627,E2 -18402.627} C_VEL
LIN {X 0,Y 258.203,Z 281.62,A -85,B 0,C 180,E1 -18404.295,E2 -18404.295} C_VEL
LIN {X 0,Y 257.168,Z 282.625,A -85,B 0,C 180,E1 -18405.588,E2 -18405.588} C_VEL
LIN {X 0,Y 257.08,Z 282.933,A -85,B 0,C 180,E1 -18406.027,E2 -18406.027} C_VEL
LIN {X 0,Y 256.933,Z 285.015,A -85,B 0,C 180,E1 -18408.969,E2 -18408.969} C_VEL
LIN {X 0,Y 256.442,Z 288.006,A -85,B 0,C 180,E1 -18412.921,E2 -18412.921} C_VEL
LIN {X 0,Y 255.797,Z 291.034,A -85,B 0,C 180,E1 -18416.668,E2 -18416.668} C_VEL
LIN {X 0,Y 255.237,Z 294.013,A -85,B 0,C 180,E1 -18420.289,E2 -18420.289} C_VEL
LIN {X 0,Y 255.11,Z 294.669,A -85,B 0,C 180,E1 -18421.035,E2 -18421.035} C_VEL
LIN {X 0,Y 255.933,Z 297.831,A -85,B 0,C 180,E1 -18421.27,E2 -18421.27} C_VEL
LIN {X 0,Y 259.545,Z 310.443,A -85,B 0,C 180,E1 -18422.507,E2 -18422.507} C_VEL
LIN {X 0,Y 261.851,Z 321.51,A -85,B 0,C 180,E1 -18423.747,E2 -18423.747} C_VEL
LIN {X 0,Y 263.228,Z 330.757,A -85,B 0,C 180,E1 -18424.917,E2 -18424.917} C_VEL
LIN {X 0,Y 264.015,Z 339.999,A -85,B 0,C 180,E1 -18426.236,E2 -18426.236} C_VEL
LIN {X 0,Y 264.199,Z 346.851,A -85,B 0,C 180,E1 -18427.312,E2 -18427.312} C_VEL
LIN {X 0,Y 262.31,Z 355.733,A -85,B 0,C 180,E1 -18428.796,E2 -18428.796} C_VEL
LIN {X 0,Y 260.393,Z 364.871,A -85,B 0,C 180,E1 -18430.694,E2 -18430.694} C_VEL
LIN {X 0,Y 258.775,Z 372.451,A -85,B 0,C 180,E1 -18432.618,E2 -18432.618} C_VEL
LIN {X 0,Y 257.385,Z 378.768,A -85,B 0,C 180,E1 -18434.56,E2 -18434.56} C_VEL
LIN {X 0,Y 256.151,Z 384.029,A -85,B 0,C 180,E1 -18436.514,E2 -18436.514} C_VEL
LIN {X 0,Y 255.132,Z 389.161,A -85,B 0,C 180,E1 -18438.883,E2 -18438.883} C_VEL
LIN {X 0,Y 254.485,Z 393.153,A -85,B 0,C 180,E1 -18441.264,E2 -18441.264} C_VEL
LIN {X 0,Y 254.085,Z 396.105,A -85,B 0,C 180,E1 -18443.648,E2 -18443.648} C_VEL
LIN {X 0,Y 253.96,Z 398.558,A -85,B 0,C 180,E1 -18446.827,E2 -18446.827} C_VEL
LIN {X 0,Y 254.003,Z 399.15,A -85,B 0,C 180,E1 -18448.415,E2 -18448.415} C_VEL
LIN {X 0,Y 254.043,Z 399.306,A -85,B 0,C 180,E1 -18450,E2 -18450} C_VEL
LIN {X 0,Y 254.003,Z 399.15,A -85,B 0,C 180,E1 -18451.585,E2 -18451.585} C_VEL
LIN {X 0,Y 253.959,Z 398.558,A -85,B 0,C 180,E1 -18453.173,E2 -18453.173} C_VEL
LIN {X 0,Y 254.082,Z 396.105,A -85,B 0,C 180,E1 -18456.352,E2 -18456.352} C_VEL
LIN {X 0,Y 254.485,Z 393.153,A -85,B 0,C 180,E1 -18458.736,E2 -18458.736} C_VEL
LIN {X 0,Y 255.132,Z 389.161,A -85,B 0,C 180,E1 -18461.117,E2 -18461.117} C_VEL
LIN {X 0,Y 256.151,Z 384.029,A -85,B 0,C 180,E1 -18463.486,E2 -18463.486} C_VEL
LIN {X 0,Y 257.384,Z 378.768,A -85,B 0,C 180,E1 -18465.44,E2 -18465.44} C_VEL
LIN {X 0,Y 258.794,Z 372.451,A -85,B 0,C 180,E1 -18467.381,E2 -18467.381} C_VEL
LIN {X 0,Y 260.06,Z 366.499,A -85,B 0,C 180,E1 -18468.922,E2 -18468.922} C_VEL
LIN {X 0,Y 261.434,Z 359.57,A -85,B 0,C 180,E1 -18470.455,E2 -18470.455} C_VEL
LIN {X 0,Y 263.2,Z 351.394,A -85,B 0,C 180,E1 -18471.951,E2 -18471.951} C_VEL
LIN {X 0,Y 264.222,Z 345.584,A -85,B 0,C 180,E1 -18472.892,E2 -18472.892} C_VEL
LIN {X 0,Y 263.64,Z 334.979,A -85,B 0,C 180,E1 -18474.501,E2 -18474.501} C_VEL
LIN {X 0,Y 262.62,Z 325.912,A -85,B 0,C 180,E1 -18475.709,E2 -18475.709} C_VEL
LIN {X 0,Y 260.683,Z 315.496,A -85,B 0,C 180,E1 -18476.942,E2 -18476.942} C_VEL
LIN {X 0,Y 258.054,Z 304.747,A -85,B 0,C 180,E1 -18478.057,E2 -18478.057} C_VEL
LIN {X 0,Y 255.193,Z 295.411,A -85,B 0,C 180,E1 -18478.923,E2 -18478.923} C_VEL
LIN {X 0,Y 255.111,Z 294.667,A -85,B 0,C 180,E1 -18478.997,E2 -18478.997} C_VEL
LIN {X 0,Y 255.52,Z 292.479,A -85,B 0,C 180,E1 -18481.505,E2 -18481.505} C_VEL
LIN {X 0,Y 256.096,Z 289.501,A -85,B 0,C 180,E1 -18485.19,E2 -18485.19} C_VEL
LIN {X 0,Y 256.715,Z 286.504,A -85,B 0,C 180,E1 -18489.024,E2 -18489.024} C_VEL
LIN {X 0,Y 257.061,Z 284.008,A -85,B 0,C 180,E1 -18492.414,E2 -18492.414} C_VEL
LIN {X 0,Y 257.106,Z 282.024,A -85,B 0,C 180,E1 -18495.291,E2 -18495.291} C_VEL
LIN {X 0,Y 256.879,Z 279.706,A -85,B 0,C 180,E1 -18498.948,E2 -18498.948} C_VEL
LIN {X 0,Y 256.547,Z 277.393,A -85,B 0,C 180,E1 -18502.929,E2 -18502.929} C_VEL
LIN {X 0,Y 256.264,Z 275.411,A -85,B 0,C 180,E1 -18506.727,E2 -18506.727} C_VEL
LIN {X 0,Y 256.16,Z 274.52,A -85,B 0,C 180,E1 -18508.573,E2 -18508.573} C_VEL
LIN {X 0,Y 256.097,Z 274.087,A -85,B 0,C 180,E1 -18511.419,E2 -18511.419} C_VEL
LIN {X 0,Y 256.12,Z 274.085,A -85,B 0,C 180,E1 -18515.686,E2 -18515.686} C_VEL
LIN {X 0,Y 256.13,Z 274.082,A -85,B 0,C 180,E1 -18519.093,E2 -18519.093} C_VEL
LIN {X 0,Y 256.234,Z 274.067,A -85,B 0,C 180,E1 -18524.072,E2 -18524.072} C_VEL
LIN {X 0,Y 256.288,Z 274.06,A -85,B 0,C 180,E1 -18528.924,E2 -18528.924} C_VEL
LIN {X 0,Y 256.493,Z 274.034,A -85,B 0,C 180,E1 -18532.117,E2 -18532.117} C_VEL
LIN {X 0,Y 256.45,Z 274.04,A -85,B 0,C 180,E1 -18536.849,E2 -18536.849} C_VEL
LIN {X 0,Y 256.742,Z 273.992,A -85,B 0,C 180,E1 -18539.991,E2 -18539.991} C_VEL
LIN {X 0,Y 256.482,Z 274.022,A -85,B 0,C 180,E1 -18543.132,E2 -18543.132} C_VEL
LIN {X 0,Y 256.485,Z 274.034,A -85,B 0,C 180,E1 -18547.865,E2 -18547.865} C_VEL
LIN {X 0,Y 256.238,Z 274.068,A -85,B 0,C 180,E1 -18552.665,E2 -18552.665} C_VEL
LIN {X 0,Y 256.197,Z 274.069,A -85,B 0,C 180,E1 -18556.241,E2 -18556.241} C_VEL
LIN {X 0,Y 256.101,Z 274.084,A -85,B 0,C 180,E1 -18561.09,E2 -18561.09} C_VEL
LIN {X 0,Y 256.144,Z 274.075,A -85,B 0,C 180,E1 -18565.12,E2 -18565.12} C_VEL
LIN {X 0,Y 256.086,Z 274.087,A -85,B 0,C 180,E1 -18568.576,E2 -18568.576} C_VEL
LIN {X 0,Y 256.052,Z 274.087,A -85,B 0,C 180,E1 -18573.282,E2 -18573.282} C_VEL
LIN {X 0,Y 256.104,Z 274.082,A -85,B 0,C 180,E1 -18577.269,E2 -18577.269} C_VEL
LIN {X 0,Y 256.067,Z 274.087,A -85,B 0,C 180,E1 -18581.186,E2 -18581.186} C_VEL
LIN {X 0,Y 256.077,Z 274.086,A -85,B 0,C 180,E1 -18584.476,E2 -18584.476} C_VEL
LIN {X 0,Y 256.09,Z 274.085,A -85,B 0,C 180,E1 -18587.797,E2 -18587.797} C_VEL
LIN {X 0,Y 256.065,Z 274.087,A -85,B 0,C 180,E1 -18590.858,E2 -18590.858} C_VEL
LIN {X 0,Y 256.074,Z 274.087,A -85,B 0,C 180,E1 -18594.807,E2 -18594.807} C_VEL
LIN {X 0,Y 256.043,Z 274.091,A -85,B 0,C 180,E1 -18598.567,E2 -18598.567} C_VEL
LIN {X 0,Y 256.065,Z 274.089,A -85,B 0,C 180,E1 -18600.817,E2 -18600.817} C_VEL
LIN {X 0,Y 257.173,Z 277.073,A -85,B 0,C 180,E1 -18601.067,E2 -18601.067} C_VEL
LIN {X 0,Y 262.299,Z 287.238,A -85,B 0,C 180,E1 -18602.127,E2 -18602.127} C_VEL
LIN {X 0,Y 267.663,Z 299.703,A -85,B 0,C 180,E1 -18603.569,E2 -18603.569} C_VEL
LIN {X 0,Y 271.927,Z 307.939,A -85,B 0,C 180,E1 -18604.739,E2 -18604.739} C_VEL
LIN {X 0,Y 278.026,Z 317.594,A -85,B 0,C 180,E1 -18606.367,E2 -18606.367} C_VEL
LIN {X 0,Y 285.887,Z 327.712,A -85,B 0,C 180,E1 -18608.362,E2 -18608.362} C_VEL
LIN {X 0,Y 295.63,Z 338.629,A -85,B 0,C 180,E1 -18610.805,E2 -18610.805} C_VEL
LIN {X 0,Y 304.742,Z 347.889,A -85,B 0,C 180,E1 -18613.114,E2 -18613.114} C_VEL
LIN {X 0,Y 311.214,Z 354.139,A -85,B 0,C 180,E1 -18614.841,E2 -18614.841} C_VEL
LIN {X 0,Y 316.57,Z 359.338,A -85,B 0,C 180,E1 -18616.489,E2 -18616.489} C_VEL
LIN {X 0,Y 321.149,Z 363.478,A -85,B 0,C 180,E1 -18618.002,E2 -18618.002} C_VEL
LIN {X 0,Y 324.842,Z 366.658,A -85,B 0,C 180,E1 -18619.403,E2 -18619.403} C_VEL
LIN {X 0,Y 327.681,Z 368.861,A -85,B 0,C 180,E1 -18620.543,E2 -18620.543} C_VEL
LIN {X 0,Y 330.555,Z 371.558,A -85,B 0,C 180,E1 -18622.057,E2 -18622.057} C_VEL
LIN {X 0,Y 333.527,Z 374.098,A -85,B 0,C 180,E1 -18623.952,E2 -18623.952} C_VEL
LIN {X 0,Y 335.272,Z 375.217,A -85,B 0,C 180,E1 -18625.19,E2 -18625.19} C_VEL
LIN {X 0,Y 337.678,Z 376.37,A -85,B 0,C 180,E1 -18627.225,E2 -18627.225} C_VEL
LIN {X 0,Y 338.949,Z 376.745,A -85,B 0,C 180,E1 -18628.812,E2 -18628.812} C_VEL
LIN {X 0,Y 339.316,Z 376.806,A -85,B 0,C 180,E1 -18630,E2 -18630} C_VEL
LIN {X 0,Y 338.962,Z 376.741,A -85,B 0,C 180,E1 -18631.188,E2 -18631.188} C_VEL
LIN {X 0,Y 337.674,Z 376.382,A -85,B 0,C 180,E1 -18632.762,E2 -18632.762} C_VEL
LIN {X 0,Y 335.278,Z 375.228,A -85,B 0,C 180,E1 -18634.81,E2 -18634.81} C_VEL
LIN {X 0,Y 332.529,Z 373.344,A -85,B 0,C 180,E1 -18636.705,E2 -18636.705} C_VEL
LIN {X 0,Y 329.461,Z 370.435,A -85,B 0,C 180,E1 -18638.587,E2 -18638.587} C_VEL
LIN {X 0,Y 326.585,Z 368.021,A -85,B 0,C 180,E1 -18639.913,E2 -18639.913} C_VEL
LIN {X 0,Y 321.185,Z 363.473,A -85,B 0,C 180,E1 -18641.997,E2 -18641.997} C_VEL
LIN {X 0,Y 315.461,Z 358.275,A -85,B 0,C 180,E1 -18643.877,E2 -18643.877} C_VEL
LIN {X 0,Y 309.916,Z 352.924,A -85,B 0,C 180,E1 -18645.512,E2 -18645.512} C_VEL
LIN {X 0,Y 301.889,Z 345.051,A -85,B 0,C 180,E1 -18647.616,E2 -18647.616} C_VEL
LIN {X 0,Y 293.148,Z 335.996,A -85,B 0,C 180,E1 -18649.815,E2 -18649.815} C_VEL
LIN {X 0,Y 283.234,Z 324.476,A -85,B 0,C 180,E1 -18652.305,E2 -18652.305} C_VEL
LIN {X 0,Y 276.762,Z 315.688,A -85,B 0,C 180,E1 -18653.972,E2 -18653.972} C_VEL
LIN {X 0,Y 270.712,Z 305.818,A -85,B 0,C 180,E1 -18655.586,E2 -18655.586} C_VEL
LIN {X 0,Y 266.102,Z 296.118,A -85,B 0,C 180,E1 -18656.876,E2 -18656.876} C_VEL
LIN {X 0,Y 260.411,Z 283.174,A -85,B 0,C 180,E1 -18658.298,E2 -18658.298} C_VEL
LIN {X 0,Y 256.319,Z 275.269,A -85,B 0,C 180,E1 -18659.102,E2 -18659.102} C_VEL
LIN {X 0,Y 256.066,Z 274.089,A -85,B 0,C 180,E1 -18659.184,E2 -18659.184} C_VEL
LIN {X 0,Y 256.038,Z 274.092,A -85,B 0,C 180,E1 -18663.296,E2 -18663.296} C_VEL
LIN {X 0,Y 256.092,Z 274.084,A -85,B 0,C 180,E1 -18667.284,E2 -18667.284} C_VEL
LIN {X 0,Y 256.062,Z 274.087,A -85,B 0,C 180,E1 -18671.201,E2 -18671.201} C_VEL
LIN {X 0,Y 256.076,Z 274.085,A -85,B 0,C 180,E1 -18674.491,E2 -18674.491} C_VEL
LIN {X 0,Y 256.094,Z 274.086,A -85,B 0,C 180,E1 -18677.812,E2 -18677.812} C_VEL
LIN {X 0,Y 256.073,Z 274.086,A -85,B 0,C 180,E1 -18680.873,E2 -18680.873} C_VEL
LIN {X 0,Y 256.087,Z 274.084,A -85,B 0,C 180,E1 -18684.822,E2 -18684.822} C_VEL
LIN {X 0,Y 256.052,Z 274.088,A -85,B 0,C 180,E1 -18688.58,E2 -18688.58} C_VEL
LIN {X 0,Y 256.099,Z 274.083,A -85,B 0,C 180,E1 -18692.203,E2 -18692.203} C_VEL
LIN {X 0,Y 256.116,Z 274.08,A -85,B 0,C 180,E1 -18695.706,E2 -18695.706} C_VEL
LIN {X 0,Y 256.103,Z 274.083,A -85,B 0,C 180,E1 -18699.111,E2 -18699.111} C_VEL
LIN {X 0,Y 256.212,Z 274.067,A -85,B 0,C 180,E1 -18704.09,E2 -18704.09} C_VEL
LIN {X 0,Y 256.272,Z 274.063,A -85,B 0,C 180,E1 -18708.942,E2 -18708.942} C_VEL
LIN {X 0,Y 256.485,Z 274.034,A -85,B 0,C 180,E1 -18712.135,E2 -18712.135} C_VEL
LIN {X 0,Y 256.482,Z 274.022,A -85,B 0,C 180,E1 -18716.868,E2 -18716.868} C_VEL
LIN {X 0,Y 256.742,Z 273.992,A -85,B 0,C 180,E1 -18720.009,E2 -18720.009} C_VEL
LIN {X 0,Y 256.45,Z 274.04,A -85,B 0,C 180,E1 -18723.151,E2 -18723.151} C_VEL
LIN {X 0,Y 256.493,Z 274.034,A -85,B 0,C 180,E1 -18727.883,E2 -18727.883} C_VEL
LIN {X 0,Y 256.256,Z 274.067,A -85,B 0,C 180,E1 -18732.683,E2 -18732.683} C_VEL
LIN {X 0,Y 256.22,Z 274.072,A -85,B 0,C 180,E1 -18736.258,E2 -18736.258} C_VEL
LIN {X 0,Y 256.128,Z 274.08,A -85,B 0,C 180,E1 -18741.106,E2 -18741.106} C_VEL
LIN {X 0,Y 256.114,Z 274.084,A -85,B 0,C 180,E1 -18745.106,E2 -18745.106} C_VEL
LIN {X 0,Y 256.097,Z 274.086,A -85,B 0,C 180,E1 -18748.581,E2 -18748.581} C_VEL
LIN {X 0,Y 256.184,Z 274.671,A -85,B 0,C 180,E1 -18751.743,E2 -18751.743} C_VEL
LIN {X 0,Y 256.406,Z 276.373,A -85,B 0,C 180,E1 -18755.151,E2 -18755.151} C_VEL
LIN {X 0,Y 256.729,Z 278.677,A -85,B 0,C 180,E1 -18759.307,E2 -18759.307} C_VEL
LIN {X 0,Y 257.046,Z 281.001,A -85,B 0,C 180,E1 -18763.13,E2 -18763.13} C_VEL
LIN {X 0,Y 257.08,Z 282.933,A -85,B 0,C 180,E1 -18766.027,E2 -18766.027} C_VEL
LIN {X 0,Y 256.374,Z 283.91,A -85,B 0,C 180,E1 -18767.314,E2 -18767.314} C_VEL
LIN {X 0,Y 253.37,Z 285.745,A -85,B 0,C 180,E1 -18769.395,E2 -18769.395} C_VEL
LIN {X 0,Y 249.798,Z 288.008,A -85,B 0,C 180,E1 -18771.96,E2 -18771.96} C_VEL
LIN {X 0,Y 249.332,Z 288.715,A -85,B 0,C 180,E1 -18772.855,E2 -18772.855} C_VEL
LIN {X 0,Y 248.904,Z 290.85,A -85,B 0,C 180,E1 -18775.618,E2 -18775.618} C_VEL
LIN {X 0,Y 248.291,Z 293.831,A -85,B 0,C 180,E1 -18779.37,E2 -18779.37} C_VEL
LIN {X 0,Y 248.197,Z 294.479,A -85,B 0,C 180,E1 -18780.136,E2 -18780.136} C_VEL
LIN {X 0,Y 249.049,Z 297.748,A -85,B 0,C 180,E1 -18780.404,E2 -18780.404} C_VEL
LIN {X 0,Y 252.635,Z 310.026,A -85,B 0,C 180,E1 -18781.67,E2 -18781.67} C_VEL
LIN {X 0,Y 254.811,Z 320.007,A -85,B 0,C 180,E1 -18782.823,E2 -18782.823} C_VEL
LIN {X 0,Y 256.363,Z 330.062,A -85,B 0,C 180,E1 -18784.132,E2 -18784.132} C_VEL
LIN {X 0,Y 257.242,Z 340.031,A -85,B 0,C 180,E1 -18785.608,E2 -18785.608} C_VEL
LIN {X 0,Y 257.4,Z 347.798,A -85,B 0,C 180,E1 -18786.891,E2 -18786.891} C_VEL
LIN {X 0,Y 255.688,Z 355.538,A -85,B 0,C 180,E1 -18788.219,E2 -18788.219} C_VEL
LIN {X 0,Y 253.682,Z 364.676,A -85,B 0,C 180,E1 -18790.162,E2 -18790.162} C_VEL
LIN {X 0,Y 252.424,Z 370.532,A -85,B 0,C 180,E1 -18791.641,E2 -18791.641} C_VEL
LIN {X 0,Y 250.792,Z 377.417,A -85,B 0,C 180,E1 -18793.726,E2 -18793.726} C_VEL
LIN {X 0,Y 249.718,Z 381.918,A -85,B 0,C 180,E1 -18795.328,E2 -18795.328} C_VEL
LIN {X 0,Y 248.455,Z 387.41,A -85,B 0,C 180,E1 -18797.752,E2 -18797.752} C_VEL
LIN {X 0,Y 247.631,Z 391.739,A -85,B 0,C 180,E1 -18800.196,E2 -18800.196} C_VEL
LIN {X 0,Y 247.282,Z 394.109,A -85,B 0,C 180,E1 -18801.831,E2 -18801.831} C_VEL
LIN {X 0,Y 247.008,Z 395.91,A -85,B 0,C 180,E1 -18803.465,E2 -18803.465} C_VEL
LIN {X 0,Y 246.862,Z 398.363,A -85,B 0,C 180,E1 -18806.736,E2 -18806.736} C_VEL
LIN {X 0,Y 246.913,Z 398.956,A -85,B 0,C 180,E1 -18808.369,E2 -18808.369} C_VEL
LIN {X 0,Y 246.951,Z 399.112,A -85,B 0,C 180,E1 -18810,E2 -18810} C_VEL
LIN {X 0,Y 246.913,Z 398.956,A -85,B 0,C 180,E1 -18811.631,E2 -18811.631} C_VEL
LIN {X 0,Y 246.861,Z 398.363,A -85,B 0,C 180,E1 -18813.264,E2 -18813.264} C_VEL
LIN {X 0,Y 247.005,Z 395.91,A -85,B 0,C 180,E1 -18816.535,E2 -18816.535} C_VEL
LIN {X 0,Y 247.43,Z 392.957,A -85,B 0,C 180,E1 -18818.987,E2 -18818.987} C_VEL
LIN {X 0,Y 248.145,Z 388.965,A -85,B 0,C 180,E1 -18821.435,E2 -18821.435} C_VEL
LIN {X 0,Y 249.221,Z 383.833,A -85,B 0,C 180,E1 -18823.868,E2 -18823.868} C_VEL
LIN {X 0,Y 250.525,Z 378.573,A -85,B 0,C 180,E1 -18825.873,E2 -18825.873} C_VEL
LIN {X 0,Y 252.025,Z 372.257,A -85,B 0,C 180,E1 -18827.863,E2 -18827.863} C_VEL
LIN {X 0,Y 253.306,Z 366.303,A -85,B 0,C 180,E1 -18829.447,E2 -18829.447} C_VEL
LIN {X 0,Y 254.768,Z 359.375,A -85,B 0,C 180,E1 -18831.015,E2 -18831.015} C_VEL
LIN {X 0,Y 256.628,Z 351.199,A -85,B 0,C 180,E1 -18832.544,E2 -18832.544} C_VEL
LIN {X 0,Y 257.474,Z 346.65,A -85,B 0,C 180,E1 -18833.315,E2 -18833.315} C_VEL
LIN {X 0,Y 256.847,Z 335.062,A -85,B 0,C 180,E1 -18835.155,E2 -18835.155} C_VEL
LIN {X 0,Y 255.871,Z 326.201,A -85,B 0,C 180,E1 -18836.385,E2 -18836.385} C_VEL
LIN {X 0,Y 253.951,Z 315.908,A -85,B 0,C 180,E1 -18837.663,E2 -18837.663} C_VEL
LIN {X 0,Y 251.271,Z 305.134,A -85,B 0,C 180,E1 -18838.846,E2 -18838.846} C_VEL
LIN {X 0,Y 248.26,Z 295.307,A -85,B 0,C 180,E1 -18839.806,E2 -18839.806} C_VEL
LIN {X 0,Y 248.19,Z 294.506,A -85,B 0,C 180,E1 -18839.869,E2 -18839.869} C_VEL
LIN {X 0,Y 248.903,Z 290.833,A -85,B 0,C 180,E1 -18844.382,E2 -18844.382} C_VEL
LIN {X 0,Y 249.545,Z 287.842,A -85,B 0,C 180,E1 -18848.285,E2 -18848.285} C_VEL
LIN {X 0,Y 249.828,Z 286.156,A -85,B 0,C 180,E1 -18850.565,E2 -18850.565} C_VEL
LIN {X 0,Y 250.059,Z 284.428,A -85,B 0,C 180,E1 -18853.041,E2 -18853.041} C_VEL
LIN {X 0,Y 250.021,Z 281.881,A -85,B 0,C 180,E1 -18856.956,E2 -18856.956} C_VEL
LIN {X 0,Y 249.781,Z 280.257,A -85,B 0,C 180,E1 -18859.664,E2 -18859.664} C_VEL
LIN {X 0,Y 249.446,Z 278.01,A -85,B 0,C 180,E1 -18863.716,E2 -18863.716} C_VEL
LIN {X 0,Y 249.18,Z 275.989,A -85,B 0,C 180,E1 -18867.792,E2 -18867.792} C_VEL
LIN {X 0,Y 249.064,Z 275.224,A -85,B 0,C 180,E1 -18869.466,E2 -18869.466} C_VEL
LIN {X 0,Y 249.033,Z 274.965,A -85,B 0,C 180,E1 -18873.149,E2 -18873.149} C_VEL
LIN {X 0,Y 249.029,Z 274.966,A -85,B 0,C 180,E1 -18876.719,E2 -18876.719} C_VEL
LIN {X 0,Y 249.064,Z 274.962,A -85,B 0,C 180,E1 -18880.199,E2 -18880.199} C_VEL
LIN {X 0,Y 249.163,Z 274.95,A -85,B 0,C 180,E1 -18883.608,E2 -18883.608} C_VEL
LIN {X 0,Y 249.188,Z 274.944,A -85,B 0,C 180,E1 -18886.951,E2 -18886.951} C_VEL
LIN {X 0,Y 249.38,Z 274.92,A -85,B 0,C 180,E1 -18890.52,E2 -18890.52} C_VEL
LIN {X 0,Y 249.432,Z 274.916,A -85,B 0,C 180,E1 -18893.52,E2 -18893.52} C_VEL
LIN {X 0,Y 249.656,Z 274.883,A -85,B 0,C 180,E1 -18898.378,E2 -18898.378} C_VEL
LIN {X 0,Y 249.665,Z 274.864,A -85,B 0,C 180,E1 -18901.604,E2 -18901.604} C_VEL
LIN {X 0,Y 249.414,Z 274.914,A -85,B 0,C 180,E1 -18906.685,E2 -18906.685} C_VEL
LIN {X 0,Y 249.321,Z 274.923,A -85,B 0,C 180,E1 -18909.727,E2 -18909.727} C_VEL
LIN {X 0,Y 249.153,Z 274.946,A -85,B 0,C 180,E1 -18914.696,E2 -18914.696} C_VEL
LIN {X 0,Y 249.074,Z 274.958,A -85,B 0,C 180,E1 -18918.071,E2 -18918.071} C_VEL
LIN {X 0,Y 249.024,Z 274.964,A -85,B 0,C 180,E1 -18921.512,E2 -18921.512} C_VEL
LIN {X 0,Y 249.09,Z 274.953,A -85,B 0,C 180,E1 -18925.465,E2 -18925.465} C_VEL
LIN {X 0,Y 249.026,Z 274.965,A -85,B 0,C 180,E1 -18928.972,E2 -18928.972} C_VEL
LIN {X 0,Y 249.002,Z 274.97,A -85,B 0,C 180,E1 -18932.417,E2 -18932.417} C_VEL
LIN {X 0,Y 249.04,Z 274.964,A -85,B 0,C 180,E1 -18936.329,E2 -18936.329} C_VEL
LIN {X 0,Y 249.041,Z 274.964,A -85,B 0,C 180,E1 -18940.456,E2 -18940.456} C_VEL
LIN {X 0,Y 249.022,Z 274.964,A -85,B 0,C 180,E1 -18944.858,E2 -18944.858} C_VEL
LIN {X 0,Y 249.037,Z 274.962,A -85,B 0,C 180,E1 -18947.369,E2 -18947.369} C_VEL
LIN {X 0,Y 249.007,Z 274.968,A -85,B 0,C 180,E1 -18951.617,E2 -18951.617} C_VEL
LIN {X 0,Y 249.015,Z 274.968,A -85,B 0,C 180,E1 -18955.636,E2 -18955.636} C_VEL
LIN {X 0,Y 249.018,Z 275.076,A -85,B 0,C 180,E1 -18959.945,E2 -18959.945} C_VEL
LIN {X 0,Y 250.002,Z 277.768,A -85,B 0,C 180,E1 -18960.175,E2 -18960.175} C_VEL
LIN {X 0,Y 255.602,Z 288.692,A -85,B 0,C 180,E1 -18961.406,E2 -18961.406} C_VEL
LIN {X 0,Y 260.605,Z 300.433,A -85,B 0,C 180,E1 -18962.84,E2 -18962.84} C_VEL
LIN {X 0,Y 264.469,Z 308.889,A -85,B 0,C 180,E1 -18964.048,E2 -18964.048} C_VEL
LIN {X 0,Y 269.925,Z 318.196,A -85,B 0,C 180,E1 -18965.655,E2 -18965.655} C_VEL
LIN {X 0,Y 276.955,Z 327.966,A -85,B 0,C 180,E1 -18967.627,E2 -18967.627} C_VEL
LIN {X 0,Y 285.937,Z 338.399,A -85,B 0,C 180,E1 -18970.039,E2 -18970.039} C_VEL
LIN {X 0,Y 294.863,Z 347.542,A -85,B 0,C 180,E1 -18972.401,E2 -18972.401} C_VEL
LIN {X 0,Y 302.584,Z 354.979,A -85,B 0,C 180,E1 -18974.517,E2 -18974.517} C_VEL
LIN {X 0,Y 307.1,Z 359.119,A -85,B 0,C 180,E1 -18975.801,E2 -18975.801} C_VEL
LIN {X 0,Y 313.051,Z 364.594,A -85,B 0,C 180,E1 -18977.686,E2 -18977.686} C_VEL
LIN {X 0,Y 317.188,Z 368.345,A -85,B 0,C 180,E1 -18979.199,E2 -18979.199} C_VEL
LIN {X 0,Y 320.593,Z 371.01,A -85,B 0,C 180,E1 -18980.503,E2 -18980.503} C_VEL
LIN {X 0,Y 323.396,Z 373.512,A -85,B 0,C 180,E1 -18981.88,E2 -18981.88} C_VEL
LIN {X 0,Y 326.515,Z 376.235,A -85,B 0,C 180,E1 -18983.822,E2 -18983.822} C_VEL
LIN {X 0,Y 328.331,Z 377.539,A -85,B 0,C 180,E1 -18985.088,E2 -18985.088} C_VEL
LIN {X 0,Y 330.716,Z 378.802,A -85,B 0,C 180,E1 -18986.973,E2 -18986.973} C_VEL
LIN {X 0,Y 332.3,Z 379.332,A -85,B 0,C 180,E1 -18988.788,E2 -18988.788} C_VEL
LIN {X 0,Y 332.706,Z 379.411,A -85,B 0,C 180,E1 -18990,E2 -18990} C_VEL
LIN {X 0,Y 332.305,Z 379.33,A -85,B 0,C 180,E1 -18991.212,E2 -18991.212} C_VEL
LIN {X 0,Y 330.708,Z 378.822,A -85,B 0,C 180,E1 -18993.001,E2 -18993.001} C_VEL
LIN {X 0,Y 328.351,Z 377.541,A -85,B 0,C 180,E1 -18994.911,E2 -18994.911} C_VEL
LIN {X 0,Y 325.531,Z 375.447,A -85,B 0,C 180,E1 -18996.821,E2 -18996.821} C_VEL
LIN {X 0,Y 323.423,Z 373.52,A -85,B 0,C 180,E1 -18998.12,E2 -18998.12} C_VEL
LIN {X 0,Y 320.582,Z 371.032,A -85,B 0,C 180,E1 -18999.485,E2 -18999.485} C_VEL
LIN {X 0,Y 315.182,Z 366.516,A -85,B 0,C 180,E1 -19001.577,E2 -19001.577} C_VEL
LIN {X 0,Y 308.873,Z 360.815,A -85,B 0,C 180,E1 -19003.659,E2 -19003.659} C_VEL
LIN {X 0,Y 302.605,Z 354.912,A -85,B 0,C 180,E1 -19005.498,E2 -19005.498} C_VEL
LIN {X 0,Y 293.704,Z 346.381,A -85,B 0,C 180,E1 -19007.907,E2 -19007.907} C_VEL
LIN {X 0,Y 284.696,Z 336.983,A -85,B 0,C 180,E1 -19010.304,E2 -19010.304} C_VEL
LIN {X 0,Y 275.98,Z 326.704,A -85,B 0,C 180,E1 -19012.643,E2 -19012.643} C_VEL
LIN {X 0,Y 269.183,Z 317.102,A -85,B 0,C 180,E1 -19014.55,E2 -19014.55} C_VEL
LIN {X 0,Y 263.74,Z 307.47,A -85,B 0,C 180,E1 -19016.173,E2 -19016.173} C_VEL
LIN {X 0,Y 259.361,Z 297.426,A -85,B 0,C 180,E1 -19017.551,E2 -19017.551} C_VEL
LIN {X 0,Y 253.779,Z 284.782,A -85,B 0,C 180,E1 -19019.036,E2 -19019.036} C_VEL
LIN {X 0,Y 249.232,Z 276.048,A -85,B 0,C 180,E1 -19019.994,E2 -19019.994} C_VEL
LIN {X 0,Y 249.007,Z 274.969,A -85,B 0,C 180,E1 -19020.082,E2 -19020.082} C_VEL
LIN {X 0,Y 249.015,Z 274.968,A -85,B 0,C 180,E1 -19024.364,E2 -19024.364} C_VEL
LIN {X 0,Y 249.007,Z 274.968,A -85,B 0,C 180,E1 -19028.383,E2 -19028.383} C_VEL
LIN {X 0,Y 249.037,Z 274.962,A -85,B 0,C 180,E1 -19032.631,E2 -19032.631} C_VEL
LIN {X 0,Y 249.04,Z 274.963,A -85,B 0,C 180,E1 -19037.384,E2 -19037.384} C_VEL
LIN {X 0,Y 249.017,Z 274.967,A -85,B 0,C 180,E1 -19041.633,E2 -19041.633} C_VEL
LIN {X 0,Y 249.029,Z 274.966,A -85,B 0,C 180,E1 -19045.651,E2 -19045.651} C_VEL
LIN {X 0,Y 248.977,Z 274.972,A -85,B 0,C 180,E1 -19049.476,E2 -19049.476} C_VEL
LIN {X 0,Y 249.036,Z 274.965,A -85,B 0,C 180,E1 -19053.17,E2 -19053.17} C_VEL
LIN {X 0,Y 249.033,Z 274.962,A -85,B 0,C 180,E1 -19056.74,E2 -19056.74} C_VEL
LIN {X 0,Y 249.037,Z 274.957,A -85,B 0,C 180,E1 -19060.217,E2 -19060.217} C_VEL
LIN {X 0,Y 249.14,Z 274.949,A -85,B 0,C 180,E1 -19063.626,E2 -19063.626} C_VEL
LIN {X 0,Y 249.215,Z 274.942,A -85,B 0,C 180,E1 -19068.625,E2 -19068.625} C_VEL
LIN {X 0,Y 249.425,Z 274.913,A -85,B 0,C 180,E1 -19071.911,E2 -19071.911} C_VEL
LIN {X 0,Y 249.273,Z 274.929,A -85,B 0,C 180,E1 -19075.158,E2 -19075.158} C_VEL
LIN {X 0,Y 249.665,Z 274.864,A -85,B 0,C 180,E1 -19078.396,E2 -19078.396} C_VEL
LIN {X 0,Y 249.656,Z 274.883,A -85,B 0,C 180,E1 -19081.622,E2 -19081.622} C_VEL
LIN {X 0,Y 249.432,Z 274.916,A -85,B 0,C 180,E1 -19086.48,E2 -19086.48} C_VEL
LIN {X 0,Y 249.334,Z 274.926,A -85,B 0,C 180,E1 -19089.746,E2 -19089.746} C_VEL
LIN {X 0,Y 249.175,Z 274.949,A -85,B 0,C 180,E1 -19094.714,E2 -19094.714} C_VEL
LIN {X 0,Y 249.1,Z 274.958,A -85,B 0,C 180,E1 -19098.089,E2 -19098.089} C_VEL
LIN {X 0,Y 249.051,Z 274.962,A -85,B 0,C 180,E1 -19101.53,E2 -19101.53} C_VEL
LIN {X 0,Y 249.071,Z 274.962,A -85,B 0,C 180,E1 -19105.456,E2 -19105.456} C_VEL
LIN {X 0,Y 249.045,Z 274.964,A -85,B 0,C 180,E1 -19108.979,E2 -19108.979} C_VEL
LIN {X 0,Y 249.064,Z 275.223,A -85,B 0,C 180,E1 -19110.534,E2 -19110.534} C_VEL
LIN {X 0,Y 249.386,Z 277.457,A -85,B 0,C 180,E1 -19115.191,E2 -19115.191} C_VEL
LIN {X 0,Y 249.6,Z 279.103,A -85,B 0,C 180,E1 -19118.286,E2 -19118.286} C_VEL
LIN {X 0,Y 249.96,Z 281.519,A -85,B 0,C 180,E1 -19122.448,E2 -19122.448} C_VEL
LIN {X 0,Y 250.055,Z 283.787,A -85,B 0,C 180,E1 -19125.986,E2 -19125.986} C_VEL
LIN {X 0,Y 249.832,Z 286.369,A -85,B 0,C 180,E1 -19129.685,E2 -19129.685} C_VEL
LIN {X 0,Y 249.332,Z 288.715,A -85,B 0,C 180,E1 -19132.855,E2 -19132.855} C_VEL
LIN {X 0,Y 248.492,Z 289.452,A -85,B 0,C 180,E1 -19133.731,E2 -19133.731} C_VEL
LIN {X 0,Y 245.398,Z 290.776,A -85,B 0,C 180,E1 -19135.084,E2 -19135.084} C_VEL
LIN {X 0,Y 242.319,Z 292.113,A -85,B 0,C 180,E1 -19136.467,E2 -19136.467} C_VEL
LIN {X 0,Y 241.538,Z 292.876,A -85,B 0,C 180,E1 -19137.379,E2 -19137.379} C_VEL
LIN {X 0,Y 241.262,Z 294.459,A -85,B 0,C 180,E1 -19139.209,E2 -19139.209} C_VEL
LIN {X 0,Y 242.176,Z 297.642,A -85,B 0,C 180,E1 -19139.482,E2 -19139.482} C_VEL
LIN {X 0,Y 246.075,Z 311.04,A -85,B 0,C 180,E1 -19140.954,E2 -19140.954} C_VEL
LIN {X 0,Y 248.199,Z 320.899,A -85,B 0,C 180,E1 -19142.161,E2 -19142.161} C_VEL
LIN {X 0,Y 249.757,Z 331.152,A -85,B 0,C 180,E1 -19143.573,E2 -19143.573} C_VEL
LIN {X 0,Y 250.456,Z 339.639,A -85,B 0,C 180,E1 -19144.871,E2 -19144.871} C_VEL
LIN {X 0,Y 250.72,Z 347.598,A -85,B 0,C 180,E1 -19146.238,E2 -19146.238} C_VEL
LIN {X 0,Y 249.095,Z 355.343,A -85,B 0,C 180,E1 -19147.612,E2 -19147.612} C_VEL
LIN {X 0,Y 246.992,Z 364.48,A -85,B 0,C 180,E1 -19149.601,E2 -19149.601} C_VEL
LIN {X 0,Y 245.592,Z 370.641,A -85,B 0,C 180,E1 -19151.207,E2 -19151.207} C_VEL
LIN {X 0,Y 243.941,Z 377.221,A -85,B 0,C 180,E1 -19153.256,E2 -19153.256} C_VEL
LIN {X 0,Y 242.823,Z 381.723,A -85,B 0,C 180,E1 -19154.901,E2 -19154.901} C_VEL
LIN {X 0,Y 241.482,Z 387.215,A -85,B 0,C 180,E1 -19157.392,E2 -19157.392} C_VEL
LIN {X 0,Y 240.62,Z 391.544,A -85,B 0,C 180,E1 -19159.907,E2 -19159.907} C_VEL
LIN {X 0,Y 240.229,Z 393.913,A -85,B 0,C 180,E1 -19161.589,E2 -19161.589} C_VEL
LIN {X 0,Y 239.933,Z 395.715,A -85,B 0,C 180,E1 -19163.272,E2 -19163.272} C_VEL
LIN {X 0,Y 239.768,Z 398.168,A -85,B 0,C 180,E1 -19166.639,E2 -19166.639} C_VEL
LIN {X 0,Y 239.824,Z 398.761,A -85,B 0,C 180,E1 -19168.321,E2 -19168.321} C_VEL
LIN {X 0,Y 239.862,Z 398.917,A -85,B 0,C 180,E1 -19170,E2 -19170} C_VEL
LIN {X 0,Y 239.824,Z 398.761,A -85,B 0,C 180,E1 -19171.679,E2 -19171.679} C_VEL
LIN {X 0,Y 239.79,Z 397.338,A -85,B 0,C 180,E1 -19174.715,E2 -19174.715} C_VEL
LIN {X 0,Y 239.929,Z 395.715,A -85,B 0,C 180,E1 -19176.729,E2 -19176.729} C_VEL
LIN {X 0,Y 240.396,Z 392.762,A -85,B 0,C 180,E1 -19179.253,E2 -19179.253} C_VEL
LIN {X 0,Y 241.167,Z 388.77,A -85,B 0,C 180,E1 -19181.77,E2 -19181.77} C_VEL
LIN {X 0,Y 242.306,Z 383.638,A -85,B 0,C 180,E1 -19184.272,E2 -19184.272} C_VEL
LIN {X 0,Y 243.677,Z 378.378,A -85,B 0,C 180,E1 -19186.332,E2 -19186.332} C_VEL
LIN {X 0,Y 245.265,Z 372.062,A -85,B 0,C 180,E1 -19188.373,E2 -19188.373} C_VEL
LIN {X 0,Y 246.566,Z 366.106,A -85,B 0,C 180,E1 -19190.001,E2 -19190.001} C_VEL
LIN {X 0,Y 248.144,Z 359.18,A -85,B 0,C 180,E1 -19191.603,E2 -19191.603} C_VEL
LIN {X 0,Y 250.084,Z 351.005,A -85,B 0,C 180,E1 -19193.168,E2 -19193.168} C_VEL
LIN {X 0,Y 250.69,Z 346.447,A -85,B 0,C 180,E1 -19193.985,E2 -19193.985} C_VEL
LIN {X 0,Y 250.22,Z 335.871,A -85,B 0,C 180,E1 -19195.732,E2 -19195.732} C_VEL
LIN {X 0,Y 249.099,Z 326.482,A -85,B 0,C 180,E1 -19197.105,E2 -19197.105} C_VEL
LIN {X 0,Y 247.038,Z 315.316,A -85,B 0,C 180,E1 -19198.541,E2 -19198.541} C_VEL
LIN {X 0,Y 244.204,Z 304.289,A -85,B 0,C 180,E1 -19199.805,E2 -19199.805} C_VEL
LIN {X 0,Y 241.298,Z 295.035,A -85,B 0,C 180,E1 -19200.76,E2 -19200.76} C_VEL
LIN {X 0,Y 241.222,Z 294.319,A -85,B 0,C 180,E1 -19200.835,E2 -19200.835} C_VEL
LIN {X 0,Y 242.028,Z 290.598,A -85,B 0,C 180,E1 -19205.592,E2 -19205.592} C_VEL
LIN {X 0,Y 242.633,Z 287.675,A -85,B 0,C 180,E1 -19209.585,E2 -19209.585} C_VEL
LIN {X 0,Y 243.005,Z 284.871,A -85,B 0,C 180,E1 -19213.685,E2 -19213.685} C_VEL
LIN {X 0,Y 242.987,Z 283.214,A -85,B 0,C 180,E1 -19216.308,E2 -19216.308} C_VEL
LIN {X 0,Y 242.84,Z 281.719,A -85,B 0,C 180,E1 -19218.802,E2 -19218.802} C_VEL
LIN {X 0,Y 242.504,Z 279.681,A -85,B 0,C 180,E1 -19222.502,E2 -19222.502} C_VEL
LIN {X 0,Y 242.232,Z 277.663,A -85,B 0,C 180,E1 -19226.537,E2 -19226.537} C_VEL
LIN {X 0,Y 241.993,Z 275.844,A -85,B 0,C 180,E1 -19230.604,E2 -19230.604} C_VEL
LIN {X 0,Y 242.008,Z 275.842,A -85,B 0,C 180,E1 -19234.188,E2 -19234.188} C_VEL
LIN {X 0,Y 241.996,Z 275.843,A -85,B 0,C 180,E1 -19238.328,E2 -19238.328} C_VEL
LIN {X 0,Y 242.119,Z 275.827,A -85,B 0,C 180,E1 -19243.309,E2 -19243.309} C_VEL
LIN {X 0,Y 242.166,Z 275.819,A -85,B 0,C 180,E1 -19248.27,E2 -19248.27} C_VEL
LIN {X 0,Y 242.383,Z 275.794,A -85,B 0,C 180,E1 -19251.655,E2 -19251.655} C_VEL
LIN {X 0,Y 242.403,Z 275.792,A -85,B 0,C 180,E1 -19253.331,E2 -19253.331} C_VEL
LIN {X 0,Y 242.616,Z 275.76,A -85,B 0,C 180,E1 -19258.33,E2 -19258.33} C_VEL
LIN {X 0,Y 242.625,Z 275.74,A -85,B 0,C 180,E1 -19261.65,E2 -19261.65} C_VEL
LIN {X 0,Y 242.397,Z 275.79,A -85,B 0,C 180,E1 -19266.656,E2 -19266.656} C_VEL
LIN {X 0,Y 242.248,Z 275.804,A -85,B 0,C 180,E1 -19270.014,E2 -19270.014} C_VEL
LIN {X 0,Y 242.103,Z 275.824,A -85,B 0,C 180,E1 -19275.134,E2 -19275.134} C_VEL
LIN {X 0,Y 242.011,Z 275.838,A -85,B 0,C 180,E1 -19278.618,E2 -19278.618} C_VEL
LIN {X 0,Y 241.966,Z 275.844,A -85,B 0,C 180,E1 -19282.173,E2 -19282.173} C_VEL
LIN {X 0,Y 242.042,Z 275.831,A -85,B 0,C 180,E1 -19285.828,E2 -19285.828} C_VEL
LIN {X 0,Y 241.947,Z 275.846,A -85,B 0,C 180,E1 -19289.578,E2 -19289.578} C_VEL
LIN {X 0,Y 241.958,Z 275.843,A -85,B 0,C 180,E1 -19293.482,E2 -19293.482} C_VEL
LIN {X 0,Y 241.977,Z 275.842,A -85,B 0,C 180,E1 -19297.569,E2 -19297.569} C_VEL
LIN {X 0,Y 241.957,Z 275.847,A -85,B 0,C 180,E1 -19301.902,E2 -19301.902} C_VEL
LIN {X 0,Y 241.967,Z 275.844,A -85,B 0,C 180,E1 -19305.808,E2 -19305.808} C_VEL
LIN {X 0,Y 241.965,Z 275.846,A -85,B 0,C 180,E1 -19310.284,E2 -19310.284} C_VEL
LIN {X 0,Y 241.992,Z 275.842,A -85,B 0,C 180,E1 -19314.491,E2 -19314.491} C_VEL
LIN {X 0,Y 241.946,Z 275.848,A -85,B 0,C 180,E1 -19318.961,E2 -19318.961} C_VEL
LIN {X 0,Y 243.069,Z 278.886,A -85,B 0,C 180,E1 -19319.275,E2 -19319.275} C_VEL
LIN {X 0,Y 248.785,Z 289.878,A -85,B 0,C 180,E1 -19320.612,E2 -19320.612} C_VEL
LIN {X 0,Y 253.434,Z 300.797,A -85,B 0,C 180,E1 -19322.018,E2 -19322.018} C_VEL
LIN {X 0,Y 257.114,Z 309.605,A -85,B 0,C 180,E1 -19323.302,E2 -19323.302} C_VEL
LIN {X 0,Y 261.73,Z 318.496,A -85,B 0,C 180,E1 -19324.849,E2 -19324.849} C_VEL
LIN {X 0,Y 268.209,Z 328.216,A -85,B 0,C 180,E1 -19326.856,E2 -19326.856} C_VEL
LIN {X 0,Y 275.986,Z 337.734,A -85,B 0,C 180,E1 -19329.114,E2 -19329.114} C_VEL
LIN {X 0,Y 285.014,Z 347.218,A -85,B 0,C 180,E1 -19331.647,E2 -19331.647} C_VEL
LIN {X 0,Y 293.901,Z 355.584,A -85,B 0,C 180,E1 -19334.138,E2 -19334.138} C_VEL
LIN {X 0,Y 299.924,Z 360.908,A -85,B 0,C 180,E1 -19335.882,E2 -19335.882} C_VEL
LIN {X 0,Y 306.816,Z 367.087,A -85,B 0,C 180,E1 -19338.103,E2 -19338.103} C_VEL
LIN {X 0,Y 312.467,Z 371.957,A -85,B 0,C 180,E1 -19340.197,E2 -19340.197} C_VEL
LIN {X 0,Y 315.92,Z 374.832,A -85,B 0,C 180,E1 -19341.686,E2 -19341.686} C_VEL
LIN {X 0,Y 319.276,Z 377.775,A -85,B 0,C 180,E1 -19343.681,E2 -19343.681} C_VEL
LIN {X 0,Y 321.174,Z 379.266,A -85,B 0,C 180,E1 -19344.979,E2 -19344.979} C_VEL
LIN {X 0,Y 323.704,Z 380.719,A -85,B 0,C 180,E1 -19346.889,E2 -19346.889} C_VEL
LIN {X 0,Y 325.417,Z 381.319,A -85,B 0,C 180,E1 -19348.763,E2 -19348.763} C_VEL
LIN {X 0,Y 325.898,Z 381.395,A -85,B 0,C 180,E1 -19350,E2 -19350} C_VEL
LIN {X 0,Y 325.414,Z 381.32,A -85,B 0,C 180,E1 -19351.237,E2 -19351.237} C_VEL
LIN {X 0,Y 323.694,Z 380.745,A -85,B 0,C 180,E1 -19353.079,E2 -19353.079} C_VEL
LIN {X 0,Y 321.172,Z 379.261,A -85,B 0,C 180,E1 -19355.021,E2 -19355.021} C_VEL
LIN {X 0,Y 318.463,Z 377.114,A -85,B 0,C 180,E1 -19356.835,E2 -19356.835} C_VEL
LIN {X 0,Y 315.933,Z 374.835,A -85,B 0,C 180,E1 -19358.314,E2 -19358.314} C_VEL
LIN {X 0,Y 312.469,Z 371.978,A -85,B 0,C 180,E1 -19359.799,E2 -19359.799} C_VEL
LIN {X 0,Y 306.849,Z 367.086,A -85,B 0,C 180,E1 -19361.896,E2 -19361.896} C_VEL
LIN {X 0,Y 299.934,Z 360.934,A -85,B 0,C 180,E1 -19364.111,E2 -19364.111} C_VEL
LIN {X 0,Y 291.479,Z 353.344,A -85,B 0,C 180,E1 -19366.55,E2 -19366.55} C_VEL
LIN {X 0,Y 282.485,Z 344.699,A -85,B 0,C 180,E1 -19369.055,E2 -19369.055} C_VEL
LIN {X 0,Y 273.681,Z 335.049,A -85,B 0,C 180,E1 -19371.548,E2 -19371.548} C_VEL
LIN {X 0,Y 266.28,Z 325.55,A -85,B 0,C 180,E1 -19373.727,E2 -19373.727} C_VEL
LIN {X 0,Y 260.458,Z 316.184,A -85,B 0,C 180,E1 -19375.577,E2 -19375.577} C_VEL
LIN {X 0,Y 255.77,Z 306.68,A -85,B 0,C 180,E1 -19377.159,E2 -19377.159} C_VEL
LIN {X 0,Y 250.561,Z 293.726,A -85,B 0,C 180,E1 -19378.903,E2 -19378.903} C_VEL
LIN {X 0,Y 244.989,Z 282.347,A -85,B 0,C 180,E1 -19380.321,E2 -19380.321} C_VEL
LIN {X 0,Y 242.182,Z 276.969,A -85,B 0,C 180,E1 -19380.937,E2 -19380.937} C_VEL
LIN {X 0,Y 241.946,Z 275.848,A -85,B 0,C 180,E1 -19381.039,E2 -19381.039} C_VEL
LIN {X 0,Y 241.984,Z 275.843,A -85,B 0,C 180,E1 -19385.611,E2 -19385.611} C_VEL
LIN {X 0,Y 241.965,Z 275.846,A -85,B 0,C 180,E1 -19389.716,E2 -19389.716} C_VEL
LIN {X 0,Y 241.967,Z 275.844,A -85,B 0,C 180,E1 -19394.192,E2 -19394.192} C_VEL
LIN {X 0,Y 241.957,Z 275.847,A -85,B 0,C 180,E1 -19398.098,E2 -19398.098} C_VEL
LIN {X 0,Y 241.977,Z 275.842,A -85,B 0,C 180,E1 -19402.431,E2 -19402.431} C_VEL
LIN {X 0,Y 241.958,Z 275.843,A -85,B 0,C 180,E1 -19406.518,E2 -19406.518} C_VEL
LIN {X 0,Y 241.957,Z 275.845,A -85,B 0,C 180,E1 -19410.619,E2 -19410.619} C_VEL
LIN {X 0,Y 242.043,Z 275.831,A -85,B 0,C 180,E1 -19414.193,E2 -19414.193} C_VEL
LIN {X 0,Y 241.971,Z 275.842,A -85,B 0,C 180,E1 -19418.343,E2 -19418.343} C_VEL
LIN {X 0,Y 242.095,Z 275.828,A -85,B 0,C 180,E1 -19423.328,E2 -19423.328} C_VEL
LIN {X 0,Y 242.149,Z 275.821,A -85,B 0,C 180,E1 -19428.289,E2 -19428.289} C_VEL
LIN {X 0,Y 242.373,Z 275.792,A -85,B 0,C 180,E1 -19431.674,E2 -19431.674} C_VEL
LIN {X 0,Y 242.233,Z 275.806,A -85,B 0,C 180,E1 -19435.017,E2 -19435.017} C_VEL
LIN {X 0,Y 242.625,Z 275.74,A -85,B 0,C 180,E1 -19438.35,E2 -19438.35} C_VEL
LIN {X 0,Y 242.616,Z 275.76,A -85,B 0,C 180,E1 -19441.67,E2 -19441.67} C_VEL
LIN {X 0,Y 242.403,Z 275.791,A -85,B 0,C 180,E1 -19446.669,E2 -19446.669} C_VEL
LIN {X 0,Y 242.263,Z 275.808,A -85,B 0,C 180,E1 -19450.033,E2 -19450.033} C_VEL
LIN {X 0,Y 242.125,Z 275.825,A -85,B 0,C 180,E1 -19455.153,E2 -19455.153} C_VEL
LIN {X 0,Y 242.036,Z 275.837,A -85,B 0,C 180,E1 -19458.636,E2 -19458.636} C_VEL
LIN {X 0,Y 241.984,Z 275.844,A -85,B 0,C 180,E1 -19462.192,E2 -19462.192} C_VEL
LIN {X 0,Y 242.001,Z 275.844,A -85,B 0,C 180,E1 -19465.834,E2 -19465.834} C_VEL
LIN {X 0,Y 241.991,Z 275.919,A -85,B 0,C 180,E1 -19469.595,E2 -19469.595} C_VEL
LIN {X 0,Y 242.232,Z 277.661,A -85,B 0,C 180,E1 -19473.463,E2 -19473.463} C_VEL
LIN {X 0,Y 242.504,Z 279.701,A -85,B 0,C 180,E1 -19477.498,E2 -19477.498} C_VEL
LIN {X 0,Y 242.867,Z 282.047,A -85,B 0,C 180,E1 -19481.736,E2 -19481.736} C_VEL
LIN {X 0,Y 242.994,Z 283.385,A -85,B 0,C 180,E1 -19483.969,E2 -19483.969} C_VEL
LIN {X 0,Y 243.006,Z 284.896,A -85,B 0,C 180,E1 -19486.315,E2 -19486.315} C_VEL
LIN {X 0,Y 242.635,Z 287.692,A -85,B 0,C 180,E1 -19490.415,E2 -19490.415} C_VEL
LIN {X 0,Y 241.996,Z 290.675,A -85,B 0,C 180,E1 -19494.492,E2 -19494.492} C_VEL
LIN {X 0,Y 241.538,Z 292.876,A -85,B 0,C 180,E1 -19497.379,E2 -19497.379} C_VEL
LIN {X 0,Y 241.451,Z 294.362,A -85,B 0,C 180,E1 -19498.185,E2 -19498.185} C_VEL
LIN {X 0,Y 241.359,Z 296.947,A -85,B 0,C 180,E1 -19498.837,E2 -19498.837} C_VEL
LIN {X 0,Y 241.184,Z 301.985,A -85,B 0,C 180,E1 -19499.565,E2 -19499.565} C_VEL
LIN {X 0,Y 241.089,Z 318.155,A -85,B 0,C 180,E1 -19500.974,E2 -19500.974} C_VEL
LIN {X 0,Y 241.288,Z 320.051,A -85,B 0,C 180,E1 -19501.216,E2 -19501.216} C_VEL
LIN {X 0,Y 242.861,Z 330.034,A -85,B 0,C 180,E1 -19502.632,E2 -19502.632} C_VEL
LIN {X 0,Y 243.711,Z 339.047,A -85,B 0,C 180,E1 -19504.06,E2 -19504.06} C_VEL
LIN {X 0,Y 243.961,Z 348.537,A -85,B 0,C 180,E1 -19505.764,E2 -19505.764} C_VEL
LIN {X 0,Y 242.049,Z 357.067,A -85,B 0,C 180,E1 -19507.374,E2 -19507.374} C_VEL
LIN {X 0,Y 240.311,Z 364.285,A -85,B 0,C 180,E1 -19509.007,E2 -19509.007} C_VEL
LIN {X 0,Y 238.773,Z 370.754,A -85,B 0,C 180,E1 -19510.749,E2 -19510.749} C_VEL
LIN {X 0,Y 237.098,Z 377.025,A -85,B 0,C 180,E1 -19512.758,E2 -19512.758} C_VEL
LIN {X 0,Y 235.945,Z 381.527,A -85,B 0,C 180,E1 -19514.45,E2 -19514.45} C_VEL
LIN {X 0,Y 234.527,Z 387.019,A -85,B 0,C 180,E1 -19517.012,E2 -19517.012} C_VEL
LIN {X 0,Y 233.594,Z 391.348,A -85,B 0,C 180,E1 -19519.6,E2 -19519.6} C_VEL
LIN {X 0,Y 233.197,Z 393.718,A -85,B 0,C 180,E1 -19521.333,E2 -19521.333} C_VEL
LIN {X 0,Y 232.714,Z 396.911,A -85,B 0,C 180,E1 -19524.802,E2 -19524.802} C_VEL
LIN {X 0,Y 232.676,Z 397.973,A -85,B 0,C 180,E1 -19526.537,E2 -19526.537} C_VEL
LIN {X 0,Y 232.738,Z 398.567,A -85,B 0,C 180,E1 -19528.27,E2 -19528.27} C_VEL
LIN {X 0,Y 232.776,Z 398.723,A -85,B 0,C 180,E1 -19530,E2 -19530} C_VEL
LIN {X 0,Y 232.737,Z 398.567,A -85,B 0,C 180,E1 -19531.73,E2 -19531.73} C_VEL
LIN {X 0,Y 232.705,Z 397.31,A -85,B 0,C 180,E1 -19534.616,E2 -19534.616} C_VEL
LIN {X 0,Y 232.852,Z 395.519,A -85,B 0,C 180,E1 -19536.934,E2 -19536.934} C_VEL
LIN {X 0,Y 233.381,Z 392.567,A -85,B 0,C 180,E1 -19539.533,E2 -19539.533} C_VEL
LIN {X 0,Y 234.183,Z 388.574,A -85,B 0,C 180,E1 -19542.126,E2 -19542.126} C_VEL
LIN {X 0,Y 235.409,Z 383.442,A -85,B 0,C 180,E1 -19544.7,E2 -19544.7} C_VEL
LIN {X 0,Y 236.841,Z 378.182,A -85,B 0,C 180,E1 -19546.817,E2 -19546.817} C_VEL
LIN {X 0,Y 238.52,Z 371.866,A -85,B 0,C 180,E1 -19548.911,E2 -19548.911} C_VEL
LIN {X 0,Y 240.262,Z 364.283,A -85,B 0,C 180,E1 -19550.997,E2 -19550.997} C_VEL
LIN {X 0,Y 242.505,Z 355.147,A -85,B 0,C 180,E1 -19553.031,E2 -19553.031} C_VEL
LIN {X 0,Y 243.95,Z 348.537,A -85,B 0,C 180,E1 -19554.238,E2 -19554.238} C_VEL
LIN {X 0,Y 243.647,Z 337.877,A -85,B 0,C 180,E1 -19556.145,E2 -19556.145} C_VEL
LIN {X 0,Y 242.34,Z 326.252,A -85,B 0,C 180,E1 -19557.928,E2 -19557.928} C_VEL
LIN {X 0,Y 240.37,Z 315.64,A -85,B 0,C 180,E1 -19559.359,E2 -19559.359} C_VEL
LIN {X 0,Y 237.394,Z 304.338,A -85,B 0,C 180,E1 -19560.733,E2 -19560.733} C_VEL
LIN {X 0,Y 234.393,Z 294.861,A -85,B 0,C 180,E1 -19561.767,E2 -19561.767} C_VEL
LIN {X 0,Y 234.317,Z 294.123,A -85,B 0,C 180,E1 -19561.872,E2 -19561.872} C_VEL
LIN {X 0,Y 235.102,Z 290.474,A -85,B 0,C 180,E1 -19566.716,E2 -19566.716} C_VEL
LIN {X 0,Y 235.505,Z 288.799,A -85,B 0,C 180,E1 -19569.102,E2 -19569.102} C_VEL
LIN {X 0,Y 235.909,Z 286.021,A -85,B 0,C 180,E1 -19573.25,E2 -19573.25} C_VEL
LIN {X 0,Y 235.922,Z 283.865,A -85,B 0,C 180,E1 -19576.742,E2 -19576.742} C_VEL
LIN {X 0,Y 235.608,Z 281.56,A -85,B 0,C 180,E1 -19580.854,E2 -19580.854} C_VEL
LIN {X 0,Y 235.268,Z 279.261,A -85,B 0,C 180,E1 -19585.409,E2 -19585.409} C_VEL
LIN {X 0,Y 235.02,Z 277.445,A -85,B 0,C 180,E1 -19589.435,E2 -19589.435} C_VEL
LIN {X 0,Y 234.912,Z 276.725,A -85,B 0,C 180,E1 -19591.391,E2 -19591.391} C_VEL
LIN {X 0,Y 234.933,Z 276.723,A -85,B 0,C 180,E1 -19595.231,E2 -19595.231} C_VEL
LIN {X 0,Y 234.949,Z 276.72,A -85,B 0,C 180,E1 -19598.955,E2 -19598.955} C_VEL
LIN {X 0,Y 235.06,Z 276.705,A -85,B 0,C 180,E1 -19603.084,E2 -19603.084} C_VEL
LIN {X 0,Y 235.098,Z 276.701,A -85,B 0,C 180,E1 -19607.912,E2 -19607.912} C_VEL
LIN {X 0,Y 235.318,Z 276.675,A -85,B 0,C 180,E1 -19611.402,E2 -19611.402} C_VEL
LIN {X 0,Y 235.355,Z 276.669,A -85,B 0,C 180,E1 -19613.13,E2 -19613.13} C_VEL
LIN {X 0,Y 235.575,Z 276.637,A -85,B 0,C 180,E1 -19618.281,E2 -19618.281} C_VEL
LIN {X 0,Y 235.585,Z 276.615,A -85,B 0,C 180,E1 -19621.699,E2 -19621.699} C_VEL
LIN {X 0,Y 235.348,Z 276.67,A -85,B 0,C 180,E1 -19626.85,E2 -19626.85} C_VEL
LIN {X 0,Y 235.196,Z 276.683,A -85,B 0,C 180,E1 -19630.318,E2 -19630.318} C_VEL
LIN {X 0,Y 235.052,Z 276.703,A -85,B 0,C 180,E1 -19635.599,E2 -19635.599} C_VEL
LIN {X 0,Y 234.949,Z 276.713,A -85,B 0,C 180,E1 -19639.199,E2 -19639.199} C_VEL
LIN {X 0,Y 234.92,Z 276.722,A -85,B 0,C 180,E1 -19642.875,E2 -19642.875} C_VEL
LIN {X 0,Y 234.938,Z 276.721,A -85,B 0,C 180,E1 -19646.648,E2 -19646.648} C_VEL
LIN {X 0,Y 234.873,Z 276.728,A -85,B 0,C 180,E1 -19650.562,E2 -19650.562} C_VEL
LIN {X 0,Y 234.928,Z 276.722,A -85,B 0,C 180,E1 -19654.624,E2 -19654.624} C_VEL
LIN {X 0,Y 234.932,Z 276.72,A -85,B 0,C 180,E1 -19658.943,E2 -19658.943} C_VEL
LIN {X 0,Y 234.948,Z 276.718,A -85,B 0,C 180,E1 -19663.455,E2 -19663.455} C_VEL
LIN {X 0,Y 234.946,Z 276.718,A -85,B 0,C 180,E1 -19666.529,E2 -19666.529} C_VEL
LIN {X 0,Y 234.912,Z 276.723,A -85,B 0,C 180,E1 -19671.079,E2 -19671.079} C_VEL
LIN {X 0,Y 234.915,Z 276.724,A -85,B 0,C 180,E1 -19675.36,E2 -19675.36} C_VEL
LIN {X 0,Y 234.885,Z 276.752,A -85,B 0,C 180,E1 -19677.973,E2 -19677.973} C_VEL
LIN {X 0,Y 235.804,Z 279.438,A -85,B 0,C 180,E1 -19678.235,E2 -19678.235} C_VEL
LIN {X 0,Y 238.912,Z 285.016,A -85,B 0,C 180,E1 -19678.95,E2 -19678.95} C_VEL
LIN {X 0,Y 244.648,Z 296.984,A -85,B 0,C 180,E1 -19680.562,E2 -19680.562} C_VEL
LIN {X 0,Y 249.096,Z 308.371,A -85,B 0,C 180,E1 -19682.206,E2 -19682.206} C_VEL
LIN {X 0,Y 253.296,Z 317.717,A -85,B 0,C 180,E1 -19683.814,E2 -19683.814} C_VEL
LIN {X 0,Y 258.608,Z 326.79,A -85,B 0,C 180,E1 -19685.676,E2 -19685.676} C_VEL
LIN {X 0,Y 265.431,Z 336.141,A -85,B 0,C 180,E1 -19687.897,E2 -19687.897} C_VEL
LIN {X 0,Y 274.139,Z 345.853,A -85,B 0,C 180,E1 -19690.533,E2 -19690.533} C_VEL
LIN {X 0,Y 284.057,Z 355.354,A -85,B 0,C 180,E1 -19693.44,E2 -19693.44} C_VEL
LIN {X 0,Y 292.015,Z 362.196,A -85,B 0,C 180,E1 -19695.799,E2 -19695.799} C_VEL
LIN {X 0,Y 298.087,Z 367.333,A -85,B 0,C 180,E1 -19697.749,E2 -19697.749} C_VEL
LIN {X 0,Y 302.477,Z 370.956,A -85,B 0,C 180,E1 -19699.288,E2 -19699.288} C_VEL
LIN {X 0,Y 308.112,Z 375.439,A -85,B 0,C 180,E1 -19701.474,E2 -19701.474} C_VEL
LIN {X 0,Y 311.348,Z 378.295,A -85,B 0,C 180,E1 -19703.221,E2 -19703.221} C_VEL
LIN {X 0,Y 313.835,Z 380.366,A -85,B 0,C 180,E1 -19704.861,E2 -19704.861} C_VEL
LIN {X 0,Y 316.654,Z 382.075,A -85,B 0,C 180,E1 -19706.93,E2 -19706.93} C_VEL
LIN {X 0,Y 318.374,Z 382.689,A -85,B 0,C 180,E1 -19708.735,E2 -19708.735} C_VEL
LIN {X 0,Y 318.929,Z 382.802,A -85,B 0,C 180,E1 -19710,E2 -19710} C_VEL
LIN {X 0,Y 318.365,Z 382.693,A -85,B 0,C 180,E1 -19711.265,E2 -19711.265} C_VEL
LIN {X 0,Y 316.645,Z 382.098,A -85,B 0,C 180,E1 -19713.041,E2 -19713.041} C_VEL
LIN {X 0,Y 313.829,Z 380.357,A -85,B 0,C 180,E1 -19715.139,E2 -19715.139} C_VEL
LIN {X 0,Y 311.348,Z 378.289,A -85,B 0,C 180,E1 -19716.778,E2 -19716.778} C_VEL
LIN {X 0,Y 308.089,Z 375.44,A -85,B 0,C 180,E1 -19718.527,E2 -19718.527} C_VEL
LIN {X 0,Y 302.524,Z 370.955,A -85,B 0,C 180,E1 -19720.71,E2 -19720.71} C_VEL
LIN {X 0,Y 296.578,Z 366.011,A -85,B 0,C 180,E1 -19722.762,E2 -19722.762} C_VEL
LIN {X 0,Y 290.518,Z 360.91,A -85,B 0,C 180,E1 -19724.659,E2 -19724.659} C_VEL
LIN {X 0,Y 282.774,Z 354.184,A -85,B 0,C 180,E1 -19726.932,E2 -19726.932} C_VEL
LIN {X 0,Y 273.535,Z 345.221,A -85,B 0,C 180,E1 -19729.648,E2 -19729.648} C_VEL
LIN {X 0,Y 265.451,Z 336.073,A -85,B 0,C 180,E1 -19732.114,E2 -19732.114} C_VEL
LIN {X 0,Y 259.751,Z 328.46,A -85,B 0,C 180,E1 -19733.944,E2 -19733.944} C_VEL
LIN {X 0,Y 254.498,Z 319.963,A -85,B 0,C 180,E1 -19735.747,E2 -19735.747} C_VEL
LIN {X 0,Y 249.796,Z 310.172,A -85,B 0,C 180,E1 -19737.505,E2 -19737.505} C_VEL
LIN {X 0,Y 244.964,Z 297.664,A -85,B 0,C 180,E1 -19739.34,E2 -19739.34} C_VEL
LIN {X 0,Y 238.59,Z 284.293,A -85,B 0,C 180,E1 -19741.136,E2 -19741.136} C_VEL
LIN {X 0,Y 235.131,Z 277.824,A -85,B 0,C 180,E1 -19741.946,E2 -19741.946} C_VEL
LIN {X 0,Y 234.884,Z 276.728,A -85,B 0,C 180,E1 -19742.078,E2 -19742.078} C_VEL
LIN {X 0,Y 234.913,Z 276.725,A -85,B 0,C 180,E1 -19746.143,E2 -19746.143} C_VEL
LIN {X 0,Y 234.924,Z 276.721,A -85,B 0,C 180,E1 -19748.959,E2 -19748.959} C_VEL
LIN {X 0,Y 234.946,Z 276.718,A -85,B 0,C 180,E1 -19753.471,E2 -19753.471} C_VEL
LIN {X 0,Y 234.948,Z 276.718,A -85,B 0,C 180,E1 -19756.545,E2 -19756.545} C_VEL
LIN {X 0,Y 234.92,Z 276.722,A -85,B 0,C 180,E1 -19761.095,E2 -19761.095} C_VEL
LIN {X 0,Y 234.928,Z 276.722,A -85,B 0,C 180,E1 -19765.376,E2 -19765.376} C_VEL
LIN {X 0,Y 234.873,Z 276.728,A -85,B 0,C 180,E1 -19769.438,E2 -19769.438} C_VEL
LIN {X 0,Y 234.967,Z 276.714,A -85,B 0,C 180,E1 -19773.805,E2 -19773.805} C_VEL
LIN {X 0,Y 234.932,Z 276.72,A -85,B 0,C 180,E1 -19778.024,E2 -19778.024} C_VEL
LIN {X 0,Y 235.036,Z 276.71,A -85,B 0,C 180,E1 -19783.104,E2 -19783.104} C_VEL
LIN {X 0,Y 235.081,Z 276.701,A -85,B 0,C 180,E1 -19787.931,E2 -19787.931} C_VEL
LIN {X 0,Y 235.307,Z 276.673,A -85,B 0,C 180,E1 -19791.422,E2 -19791.422} C_VEL
LIN {X 0,Y 235.348,Z 276.67,A -85,B 0,C 180,E1 -19793.15,E2 -19793.15} C_VEL
LIN {X 0,Y 235.585,Z 276.615,A -85,B 0,C 180,E1 -19798.301,E2 -19798.301} C_VEL
LIN {X 0,Y 235.575,Z 276.637,A -85,B 0,C 180,E1 -19801.719,E2 -19801.719} C_VEL
LIN {X 0,Y 235.355,Z 276.669,A -85,B 0,C 180,E1 -19806.87,E2 -19806.87} C_VEL
LIN {X 0,Y 235.211,Z 276.689,A -85,B 0,C 180,E1 -19810.337,E2 -19810.337} C_VEL
LIN {X 0,Y 235.075,Z 276.704,A -85,B 0,C 180,E1 -19815.618,E2 -19815.618} C_VEL
LIN {X 0,Y 234.976,Z 276.715,A -85,B 0,C 180,E1 -19819.218,E2 -19819.218} C_VEL
LIN {X 0,Y 234.931,Z 276.722,A -85,B 0,C 180,E1 -19822.895,E2 -19822.895} C_VEL
LIN {X 0,Y 234.938,Z 276.721,A -85,B 0,C 180,E1 -19826.671,E2 -19826.671} C_VEL
LIN {X 0,Y 234.912,Z 276.725,A -85,B 0,C 180,E1 -19828.609,E2 -19828.609} C_VEL
LIN {X 0,Y 235.206,Z 278.605,A -85,B 0,C 180,E1 -19833.215,E2 -19833.215} C_VEL
LIN {X 0,Y 235.395,Z 280.288,A -85,B 0,C 180,E1 -19836.674,E2 -19836.674} C_VEL
LIN {X 0,Y 235.768,Z 282.582,A -85,B 0,C 180,E1 -19840.99,E2 -19840.99} C_VEL
LIN {X 0,Y 235.929,Z 284.542,A -85,B 0,C 180,E1 -19844.364,E2 -19844.364} C_VEL
LIN {X 0,Y 235.822,Z 286.962,A -85,B 0,C 180,E1 -19848.175,E2 -19848.175} C_VEL
LIN {X 0,Y 235.489,Z 289.015,A -85,B 0,C 180,E1 -19851.192,E2 -19851.192} C_VEL
LIN {X 0,Y 234.762,Z 292.007,A -85,B 0,C 180,E1 -19855.335,E2 -19855.335} C_VEL
LIN {X 0,Y 234.361,Z 294.281,A -85,B 0,C 180,E1 -19858.2,E2 -19858.2} C_VEL
LIN {X 0,Y 235.314,Z 297.58,A -85,B 0,C 180,E1 -19858.5,E2 -19858.5} C_VEL
LIN {X 0,Y 238.848,Z 309.497,A -85,B 0,C 180,E1 -19859.863,E2 -19859.863} C_VEL
LIN {X 0,Y 241.288,Z 320.051,A -85,B 0,C 180,E1 -19861.216,E2 -19861.216} C_VEL
LIN {X 0,Y 241.53,Z 325.517,A -85,B 0,C 180,E1 -19861.877,E2 -19861.877} C_VEL
LIN {X 0,Y 239.977,Z 334.19,A -85,B 0,C 180,E1 -19862.887,E2 -19862.887} C_VEL
LIN {X 0,Y 237.872,Z 342.714,A -85,B 0,C 180,E1 -19864.016,E2 -19864.016} C_VEL
LIN {X 0,Y 237.265,Z 347.484,A -85,B 0,C 180,E1 -19864.859,E2 -19864.859} C_VEL
LIN {X 0,Y 237.092,Z 350.615,A -85,B 0,C 180,E1 -19865.482,E2 -19865.482} C_VEL
LIN {X 0,Y 234.988,Z 358.79,A -85,B 0,C 180,E1 -19867.121,E2 -19867.121} C_VEL
LIN {X 0,Y 232.677,Z 368.021,A -85,B 0,C 180,E1 -19869.405,E2 -19869.405} C_VEL
LIN {X 0,Y 230.619,Z 375.673,A -85,B 0,C 180,E1 -19871.799,E2 -19871.799} C_VEL
LIN {X 0,Y 229.091,Z 381.332,A -85,B 0,C 180,E1 -19873.973,E2 -19873.973} C_VEL
LIN {X 0,Y 227.565,Z 386.823,A -85,B 0,C 180,E1 -19876.607,E2 -19876.607} C_VEL
LIN {X 0,Y 226.59,Z 391.152,A -85,B 0,C 180,E1 -19879.275,E2 -19879.275} C_VEL
LIN {X 0,Y 226.155,Z 393.523,A -85,B 0,C 180,E1 -19881.061,E2 -19881.061} C_VEL
LIN {X 0,Y 225.805,Z 395.324,A -85,B 0,C 180,E1 -19882.848,E2 -19882.848} C_VEL
LIN {X 0,Y 225.572,Z 397.778,A -85,B 0,C 180,E1 -19886.428,E2 -19886.428} C_VEL
LIN {X 0,Y 225.634,Z 398.372,A -85,B 0,C 180,E1 -19888.215,E2 -19888.215} C_VEL
LIN {X 0,Y 225.691,Z 398.529,A -85,B 0,C 180,E1 -19890,E2 -19890} C_VEL
LIN {X 0,Y 225.634,Z 398.372,A -85,B 0,C 180,E1 -19891.785,E2 -19891.785} C_VEL
LIN {X 0,Y 225.597,Z 397.336,A -85,B 0,C 180,E1 -19894.429,E2 -19894.429} C_VEL
LIN {X 0,Y 225.799,Z 395.324,A -85,B 0,C 180,E1 -19897.152,E2 -19897.152} C_VEL
LIN {X 0,Y 226.346,Z 392.371,A -85,B 0,C 180,E1 -19899.833,E2 -19899.833} C_VEL
LIN {X 0,Y 227.197,Z 388.378,A -85,B 0,C 180,E1 -19902.505,E2 -19902.505} C_VEL
LIN {X 0,Y 228.528,Z 383.247,A -85,B 0,C 180,E1 -19905.153,E2 -19905.153} C_VEL
LIN {X 0,Y 229.999,Z 377.986,A -85,B 0,C 180,E1 -19907.333,E2 -19907.333} C_VEL
LIN {X 0,Y 231.769,Z 371.67,A -85,B 0,C 180,E1 -19909.484,E2 -19909.484} C_VEL
LIN {X 0,Y 233.218,Z 365.715,A -85,B 0,C 180,E1 -19911.199,E2 -19911.199} C_VEL
LIN {X 0,Y 234.958,Z 358.789,A -85,B 0,C 180,E1 -19912.883,E2 -19912.883} C_VEL
LIN {X 0,Y 237.042,Z 350.614,A -85,B 0,C 180,E1 -19914.524,E2 -19914.524} C_VEL
LIN {X 0,Y 237.161,Z 343.411,A -85,B 0,C 180,E1 -19915.918,E2 -19915.918} C_VEL
LIN {X 0,Y 236.69,Z 334.457,A -85,B 0,C 180,E1 -19917.468,E2 -19917.468} C_VEL
LIN {X 0,Y 235.27,Z 324.025,A -85,B 0,C 180,E1 -19919.088,E2 -19919.088} C_VEL
LIN {X 0,Y 233.515,Z 315.322,A -85,B 0,C 180,E1 -19920.32,E2 -19920.32} C_VEL
LIN {X 0,Y 230.579,Z 304.217,A -85,B 0,C 180,E1 -19921.738,E2 -19921.738} C_VEL
LIN {X 0,Y 227.916,Z 296.352,A -85,B 0,C 180,E1 -19922.697,E2 -19922.697} C_VEL
LIN {X 0,Y 227.396,Z 293.989,A -85,B 0,C 180,E1 -19922.899,E2 -19922.899} C_VEL
LIN {X 0,Y 228.035,Z 291.183,A -85,B 0,C 180,E1 -19926.732,E2 -19926.732} C_VEL
LIN {X 0,Y 228.541,Z 288.829,A -85,B 0,C 180,E1 -19930.223,E2 -19930.223} C_VEL
LIN {X 0,Y 228.793,Z 287.344,A -85,B 0,C 180,E1 -19932.514,E2 -19932.514} C_VEL
LIN {X 0,Y 228.897,Z 285.764,A -85,B 0,C 180,E1 -19935.064,E2 -19935.064} C_VEL
LIN {X 0,Y 228.863,Z 284.347,A -85,B 0,C 180,E1 -19937.49,E2 -19937.49} C_VEL
LIN {X 0,Y 228.436,Z 281.956,A -85,B 0,C 180,E1 -19942.015,E2 -19942.015} C_VEL
LIN {X 0,Y 228.22,Z 279.889,A -85,B 0,C 180,E1 -19946.327,E2 -19946.327} C_VEL
LIN {X 0,Y 227.947,Z 278.125,A -85,B 0,C 180,E1 -19950.432,E2 -19950.432} C_VEL
LIN {X 0,Y 227.915,Z 277.597,A -85,B 0,C 180,E1 -19953.409,E2 -19953.409} C_VEL
LIN {X 0,Y 227.93,Z 277.596,A -85,B 0,C 180,E1 -19958.274,E2 -19958.274} C_VEL
LIN {X 0,Y 228.022,Z 277.583,A -85,B 0,C 180,E1 -19963.886,E2 -19963.886} C_VEL
LIN {X 0,Y 228.056,Z 277.579,A -85,B 0,C 180,E1 -19967.533,E2 -19967.533} C_VEL
LIN {X 0,Y 228.256,Z 277.553,A -85,B 0,C 180,E1 -19971.134,E2 -19971.134} C_VEL
LIN {X 0,Y 228.307,Z 277.546,A -85,B 0,C 180,E1 -19972.917,E2 -19972.917} C_VEL
LIN {X 0,Y 228.533,Z 277.514,A -85,B 0,C 180,E1 -19978.228,E2 -19978.228} C_VEL
LIN {X 0,Y 228.543,Z 277.491,A -85,B 0,C 180,E1 -19981.752,E2 -19981.752} C_VEL
LIN {X 0,Y 228.3,Z 277.549,A -85,B 0,C 180,E1 -19987.062,E2 -19987.062} C_VEL
LIN {X 0,Y 228.127,Z 277.565,A -85,B 0,C 180,E1 -19990.641,E2 -19990.641} C_VEL
LIN {X 0,Y 228.014,Z 277.579,A -85,B 0,C 180,E1 -19994.264,E2 -19994.264} C_VEL
LIN {X 0,Y 227.91,Z 277.594,A -85,B 0,C 180,E1 -19997.949,E2 -19997.949} C_VEL
LIN {X 0,Y 227.876,Z 277.6,A -85,B 0,C 180,E1 -20002.299,E2 -20002.299} C_VEL
LIN {X 0,Y 227.914,Z 277.595,A -85,B 0,C 180,E1 -20006.591,E2 -20006.591} C_VEL
LIN {X 0,Y 227.848,Z 277.605,A -85,B 0,C 180,E1 -20010.272,E2 -20010.272} C_VEL
LIN {X 0,Y 227.857,Z 277.6,A -85,B 0,C 180,E1 -20013.709,E2 -20013.709} C_VEL
LIN {X 0,Y 227.837,Z 277.605,A -85,B 0,C 180,E1 -20018.076,E2 -20018.076} C_VEL
LIN {X 0,Y 227.884,Z 277.598,A -85,B 0,C 180,E1 -20022.708,E2 -20022.708} C_VEL
LIN {X 0,Y 227.881,Z 277.597,A -85,B 0,C 180,E1 -20027.275,E2 -20027.275} C_VEL
LIN {X 0,Y 227.828,Z 277.607,A -85,B 0,C 180,E1 -20031.907,E2 -20031.907} C_VEL
LIN {X 0,Y 227.844,Z 277.605,A -85,B 0,C 180,E1 -20036.367,E2 -20036.367} C_VEL
LIN {X 0,Y 227.874,Z 277.655,A -85,B 0,C 180,E1 -20036.891,E2 -20036.891} C_VEL
LIN {X 0,Y 229.02,Z 280.679,A -85,B 0,C 180,E1 -20037.228,E2 -20037.228} C_VEL
LIN {X 0,Y 233.58,Z 289.131,A -85,B 0,C 180,E1 -20038.402,E2 -20038.402} C_VEL
LIN {X 0,Y 238.467,Z 299.593,A -85,B 0,C 180,E1 -20039.934,E2 -20039.934} C_VEL
LIN {X 0,Y 242.608,Z 310.429,A -85,B 0,C 180,E1 -20041.613,E2 -20041.613} C_VEL
LIN {X 0,Y 246.138,Z 318.957,A -85,B 0,C 180,E1 -20043.133,E2 -20043.133} C_VEL
LIN {X 0,Y 251.429,Z 328.701,A -85,B 0,C 180,E1 -20045.211,E2 -20045.211} C_VEL
LIN {X 0,Y 256.919,Z 336.674,A -85,B 0,C 180,E1 -20047.178,E2 -20047.178} C_VEL
LIN {X 0,Y 264.982,Z 346.12,A -85,B 0,C 180,E1 -20049.831,E2 -20049.831} C_VEL
LIN {X 0,Y 274.721,Z 355.613,A -85,B 0,C 180,E1 -20052.858,E2 -20052.858} C_VEL
LIN {X 0,Y 283.153,Z 362.682,A -85,B 0,C 180,E1 -20055.419,E2 -20055.419} C_VEL
LIN {X 0,Y 289.279,Z 367.581,A -85,B 0,C 180,E1 -20057.37,E2 -20057.37} C_VEL
LIN {X 0,Y 293.998,Z 371.195,A -85,B 0,C 180,E1 -20058.975,E2 -20058.975} C_VEL
LIN {X 0,Y 298.924,Z 374.973,A -85,B 0,C 180,E1 -20060.845,E2 -20060.845} C_VEL
LIN {X 0,Y 301.673,Z 376.938,A -85,B 0,C 180,E1 -20061.965,E2 -20061.965} C_VEL
LIN {X 0,Y 304.249,Z 379.107,A -85,B 0,C 180,E1 -20063.368,E2 -20063.368} C_VEL
LIN {X 0,Y 306.342,Z 380.847,A -85,B 0,C 180,E1 -20064.735,E2 -20064.735} C_VEL
LIN {X 0,Y 308.269,Z 382.162,A -85,B 0,C 180,E1 -20066.078,E2 -20066.078} C_VEL
LIN {X 0,Y 309.978,Z 383.023,A -85,B 0,C 180,E1 -20067.401,E2 -20067.401} C_VEL
LIN {X 0,Y 311.213,Z 383.513,A -85,B 0,C 180,E1 -20068.706,E2 -20068.706} C_VEL
LIN {X 0,Y 311.855,Z 383.668,A -85,B 0,C 180,E1 -20070,E2 -20070} C_VEL
LIN {X 0,Y 311.199,Z 383.514,A -85,B 0,C 180,E1 -20071.294,E2 -20071.294} C_VEL
LIN {X 0,Y 309.572,Z 382.846,A -85,B 0,C 180,E1 -20072.915,E2 -20072.915} C_VEL
LIN {X 0,Y 308.245,Z 382.164,A -85,B 0,C 180,E1 -20073.922,E2 -20073.922} C_VEL
LIN {X 0,Y 306.336,Z 380.847,A -85,B 0,C 180,E1 -20075.265,E2 -20075.265} C_VEL
LIN {X 0,Y 303.048,Z 378.057,A -85,B 0,C 180,E1 -20077.327,E2 -20077.327} C_VEL
LIN {X 0,Y 301.65,Z 376.939,A -85,B 0,C 180,E1 -20078.036,E2 -20078.036} C_VEL
LIN {X 0,Y 296.104,Z 372.83,A -85,B 0,C 180,E1 -20080.254,E2 -20080.254} C_VEL
LIN {X 0,Y 291.774,Z 369.438,A -85,B 0,C 180,E1 -20081.813,E2 -20081.813} C_VEL
LIN {X 0,Y 285.769,Z 364.736,A -85,B 0,C 180,E1 -20083.78,E2 -20083.78} C_VEL
LIN {X 0,Y 277.991,Z 358.393,A -85,B 0,C 180,E1 -20086.161,E2 -20086.161} C_VEL
LIN {X 0,Y 269.86,Z 351.069,A -85,B 0,C 180,E1 -20088.636,E2 -20088.636} C_VEL
LIN {X 0,Y 260.674,Z 341.284,A -85,B 0,C 180,E1 -20091.575,E2 -20091.575} C_VEL
LIN {X 0,Y 254.608,Z 333.591,A -85,B 0,C 180,E1 -20093.61,E2 -20093.61} C_VEL
LIN {X 0,Y 248.61,Z 323.844,A -85,B 0,C 180,E1 -20095.875,E2 -20095.875} C_VEL
LIN {X 0,Y 244.316,Z 314.785,A -85,B 0,C 180,E1 -20097.648,E2 -20097.648} C_VEL
LIN {X 0,Y 239.805,Z 302.911,A -85,B 0,C 180,E1 -20099.564,E2 -20099.564} C_VEL
LIN {X 0,Y 235.631,Z 293.322,A -85,B 0,C 180,E1 -20100.988,E2 -20100.988} C_VEL
LIN {X 0,Y 230.641,Z 283.587,A -85,B 0,C 180,E1 -20102.388,E2 -20102.388} C_VEL
LIN {X 0,Y 229.143,Z 280.843,A -85,B 0,C 180,E1 -20102.76,E2 -20102.76} C_VEL
LIN {X 0,Y 227.946,Z 278.108,A -85,B 0,C 180,E1 -20103.077,E2 -20103.077} C_VEL
LIN {X 0,Y 227.857,Z 277.603,A -85,B 0,C 180,E1 -20103.162,E2 -20103.162} C_VEL
LIN {X 0,Y 227.864,Z 277.602,A -85,B 0,C 180,E1 -20106.708,E2 -20106.708} C_VEL
LIN {X 0,Y 227.853,Z 277.602,A -85,B 0,C 180,E1 -20110.37,E2 -20110.37} C_VEL
LIN {X 0,Y 227.877,Z 277.598,A -85,B 0,C 180,E1 -20114.836,E2 -20114.836} C_VEL
LIN {X 0,Y 227.881,Z 277.599,A -85,B 0,C 180,E1 -20117.745,E2 -20117.745} C_VEL
LIN {X 0,Y 227.837,Z 277.605,A -85,B 0,C 180,E1 -20121.924,E2 -20121.924} C_VEL
LIN {X 0,Y 227.858,Z 277.6,A -85,B 0,C 180,E1 -20126.384,E2 -20126.384} C_VEL
LIN {X 0,Y 227.855,Z 277.601,A -85,B 0,C 180,E1 -20130.442,E2 -20130.442} C_VEL
LIN {X 0,Y 227.899,Z 277.592,A -85,B 0,C 180,E1 -20134.435,E2 -20134.435} C_VEL
LIN {X 0,Y 227.896,Z 277.596,A -85,B 0,C 180,E1 -20138.293,E2 -20138.293} C_VEL
LIN {X 0,Y 228,Z 277.581,A -85,B 0,C 180,E1 -20143.905,E2 -20143.905} C_VEL
LIN {X 0,Y 228.038,Z 277.58,A -85,B 0,C 180,E1 -20147.553,E2 -20147.553} C_VEL
LIN {X 0,Y 228.245,Z 277.55,A -85,B 0,C 180,E1 -20151.155,E2 -20151.155} C_VEL
LIN {X 0,Y 228.3,Z 277.549,A -85,B 0,C 180,E1 -20152.938,E2 -20152.938} C_VEL
LIN {X 0,Y 228.543,Z 277.491,A -85,B 0,C 180,E1 -20158.248,E2 -20158.248} C_VEL
LIN {X 0,Y 228.533,Z 277.514,A -85,B 0,C 180,E1 -20161.772,E2 -20161.772} C_VEL
LIN {X 0,Y 228.307,Z 277.547,A -85,B 0,C 180,E1 -20167.083,E2 -20167.083} C_VEL
LIN {X 0,Y 228.142,Z 277.569,A -85,B 0,C 180,E1 -20170.661,E2 -20170.661} C_VEL
LIN {X 0,Y 228.035,Z 277.583,A -85,B 0,C 180,E1 -20174.284,E2 -20174.284} C_VEL
LIN {X 0,Y 227.935,Z 277.594,A -85,B 0,C 180,E1 -20177.968,E2 -20177.968} C_VEL
LIN {X 0,Y 227.903,Z 277.599,A -85,B 0,C 180,E1 -20182.316,E2 -20182.316} C_VEL
LIN {X 0,Y 227.915,Z 277.596,A -85,B 0,C 180,E1 -20186.591,E2 -20186.591} C_VEL
LIN {X 0,Y 227.947,Z 278.12,A -85,B 0,C 180,E1 -20189.568,E2 -20189.568} C_VEL
LIN {X 0,Y 228.215,Z 279.916,A -85,B 0,C 180,E1 -20193.751,E2 -20193.751} C_VEL
LIN {X 0,Y 228.437,Z 281.964,A -85,B 0,C 180,E1 -20197.985,E2 -20197.985} C_VEL
LIN {X 0,Y 228.661,Z 283.108,A -85,B 0,C 180,E1 -20200.21,E2 -20200.21} C_VEL
LIN {X 0,Y 228.833,Z 284.38,A -85,B 0,C 180,E1 -20202.517,E2 -20202.517} C_VEL
LIN {X 0,Y 228.897,Z 285.869,A -85,B 0,C 180,E1 -20205.076,E2 -20205.076} C_VEL
LIN {X 0,Y 228.791,Z 287.359,A -85,B 0,C 180,E1 -20207.507,E2 -20207.507} C_VEL
LIN {X 0,Y 228.49,Z 289.178,A -85,B 0,C 180,E1 -20210.272,E2 -20210.272} C_VEL
LIN {X 0,Y 227.882,Z 291.82,A -85,B 0,C 180,E1 -20214.129,E2 -20214.129} C_VEL
LIN {X 0,Y 227.429,Z 293.94,A -85,B 0,C 180,E1 -20217.1,E2 -20217.1} C_VEL
LIN {X 0,Y 228.372,Z 297.305,A -85,B 0,C 180,E1 -20217.424,E2 -20217.424} C_VEL
LIN {X 0,Y 231.991,Z 309.167,A -85,B 0,C 180,E1 -20218.863,E2 -20218.863} C_VEL
LIN {X 0,Y 234.561,Z 320.14,A -85,B 0,C 180,E1 -20220.346,E2 -20220.346} C_VEL
LIN {X 0,Y 236.098,Z 329.855,A -85,B 0,C 180,E1 -20221.784,E2 -20221.784} C_VEL
LIN {X 0,Y 237.019,Z 338.842,A -85,B 0,C 180,E1 -20223.27,E2 -20223.27} C_VEL
LIN {X 0,Y 237.265,Z 347.484,A -85,B 0,C 180,E1 -20224.859,E2 -20224.859} C_VEL
LIN {X 0,Y 236.604,Z 350.102,A -85,B 0,C 180,E1 -20225.322,E2 -20225.322} C_VEL
LIN {X 0,Y 234.38,Z 353.614,A -85,B 0,C 180,E1 -20225.82,E2 -20225.82} C_VEL
LIN {X 0,Y 228.727,Z 360.216,A -85,B 0,C 180,E1 -20226.846,E2 -20226.846} C_VEL
LIN {X 0,Y 227.281,Z 363.007,A -85,B 0,C 180,E1 -20227.481,E2 -20227.481} C_VEL
LIN {X 0,Y 225.274,Z 370.488,A -85,B 0,C 180,E1 -20229.589,E2 -20229.589} C_VEL
LIN {X 0,Y 223.494,Z 376.633,A -85,B 0,C 180,E1 -20231.672,E2 -20231.672} C_VEL
LIN {X 0,Y 222.261,Z 381.137,A -85,B 0,C 180,E1 -20233.466,E2 -20233.466} C_VEL
LIN {X 0,Y 220.627,Z 386.627,A -85,B 0,C 180,E1 -20236.178,E2 -20236.178} C_VEL
LIN {X 0,Y 219.602,Z 390.957,A -85,B 0,C 180,E1 -20238.93,E2 -20238.93} C_VEL
LIN {X 0,Y 219.106,Z 393.327,A -85,B 0,C 180,E1 -20240.771,E2 -20240.771} C_VEL
LIN {X 0,Y 218.733,Z 395.129,A -85,B 0,C 180,E1 -20242.616,E2 -20242.616} C_VEL
LIN {X 0,Y 218.477,Z 397.583,A -85,B 0,C 180,E1 -20246.311,E2 -20246.311} C_VEL
LIN {X 0,Y 218.532,Z 398.177,A -85,B 0,C 180,E1 -20248.157,E2 -20248.157} C_VEL
LIN {X 0,Y 218.608,Z 398.335,A -85,B 0,C 180,E1 -20250,E2 -20250} C_VEL
LIN {X 0,Y 218.533,Z 398.177,A -85,B 0,C 180,E1 -20251.843,E2 -20251.843} C_VEL
LIN {X 0,Y 218.508,Z 397.321,A -85,B 0,C 180,E1 -20254.291,E2 -20254.291} C_VEL
LIN {X 0,Y 218.726,Z 395.129,A -85,B 0,C 180,E1 -20257.384,E2 -20257.384} C_VEL
LIN {X 0,Y 219.332,Z 392.176,A -85,B 0,C 180,E1 -20260.15,E2 -20260.15} C_VEL
LIN {X 0,Y 220.222,Z 388.182,A -85,B 0,C 180,E1 -20262.908,E2 -20262.908} C_VEL
LIN {X 0,Y 221.668,Z 383.052,A -85,B 0,C 180,E1 -20265.634,E2 -20265.634} C_VEL
LIN {X 0,Y 223.17,Z 377.789,A -85,B 0,C 180,E1 -20267.881,E2 -20267.881} C_VEL
LIN {X 0,Y 225.057,Z 371.475,A -85,B 0,C 180,E1 -20270.09,E2 -20270.09} C_VEL
LIN {X 0,Y 227.003,Z 363.892,A -85,B 0,C 180,E1 -20272.287,E2 -20272.287} C_VEL
LIN {X 0,Y 229.485,Z 354.757,A -85,B 0,C 180,E1 -20274.42,E2 -20274.42} C_VEL
LIN {X 0,Y 230.517,Z 350.417,A -85,B 0,C 180,E1 -20275.266,E2 -20275.266} C_VEL
LIN {X 0,Y 230.462,Z 341.845,A -85,B 0,C 180,E1 -20276.975,E2 -20276.975} C_VEL
LIN {X 0,Y 230.036,Z 334.709,A -85,B 0,C 180,E1 -20278.263,E2 -20278.263} C_VEL
LIN {X 0,Y 228.59,Z 324.222,A -85,B 0,C 180,E1 -20279.972,E2 -20279.972} C_VEL
LIN {X 0,Y 226.543,Z 314.323,A -85,B 0,C 180,E1 -20281.434,E2 -20281.434} C_VEL
LIN {X 0,Y 223.714,Z 303.984,A -85,B 0,C 180,E1 -20282.832,E2 -20282.832} C_VEL
LIN {X 0,Y 221.088,Z 296.362,A -85,B 0,C 180,E1 -20283.829,E2 -20283.829} C_VEL
LIN {X 0,Y 220.505,Z 293.753,A -85,B 0,C 180,E1 -20284.14,E2 -20284.14} C_VEL
LIN {X 0,Y 221.041,Z 291.488,A -85,B 0,C 180,E1 -20287.344,E2 -20287.344} C_VEL
LIN {X 0,Y 221.498,Z 289.511,A -85,B 0,C 180,E1 -20290.391,E2 -20290.391} C_VEL
LIN {X 0,Y 221.775,Z 287.163,A -85,B 0,C 180,E1 -20294.199,E2 -20294.199} C_VEL
LIN {X 0,Y 221.729,Z 284.858,A -85,B 0,C 180,E1 -20298.259,E2 -20298.259} C_VEL
LIN {X 0,Y 221.35,Z 282.529,A -85,B 0,C 180,E1 -20302.885,E2 -20302.885} C_VEL
LIN {X 0,Y 221.092,Z 280.518,A -85,B 0,C 180,E1 -20307.279,E2 -20307.279} C_VEL
LIN {X 0,Y 220.838,Z 278.828,A -85,B 0,C 180,E1 -20311.476,E2 -20311.476} C_VEL
LIN {X 0,Y 220.869,Z 278.474,A -85,B 0,C 180,E1 -20313.536,E2 -20313.536} C_VEL
LIN {X 0,Y 220.863,Z 278.477,A -85,B 0,C 180,E1 -20317.542,E2 -20317.542} C_VEL
LIN {X 0,Y 220.927,Z 278.465,A -85,B 0,C 180,E1 -20322.615,E2 -20322.615} C_VEL
LIN {X 0,Y 220.994,Z 278.457,A -85,B 0,C 180,E1 -20327.127,E2 -20327.127} C_VEL
LIN {X 0,Y 221.196,Z 278.431,A -85,B 0,C 180,E1 -20330.849,E2 -20330.849} C_VEL
LIN {X 0,Y 221.244,Z 278.425,A -85,B 0,C 180,E1 -20332.69,E2 -20332.69} C_VEL
LIN {X 0,Y 221.466,Z 278.394,A -85,B 0,C 180,E1 -20338.171,E2 -20338.171} C_VEL
LIN {X 0,Y 221.501,Z 278.367,A -85,B 0,C 180,E1 -20341.808,E2 -20341.808} C_VEL
LIN {X 0,Y 221.236,Z 278.427,A -85,B 0,C 180,E1 -20347.289,E2 -20347.289} C_VEL
LIN {X 0,Y 221.047,Z 278.449,A -85,B 0,C 180,E1 -20350.986,E2 -20350.986} C_VEL
LIN {X 0,Y 220.958,Z 278.461,A -85,B 0,C 180,E1 -20356.622,E2 -20356.622} C_VEL
LIN {X 0,Y 220.83,Z 278.471,A -85,B 0,C 180,E1 -20360.479,E2 -20360.479} C_VEL
LIN {X 0,Y 220.835,Z 278.472,A -85,B 0,C 180,E1 -20364.425,E2 -20364.425} C_VEL
LIN {X 0,Y 220.786,Z 278.483,A -85,B 0,C 180,E1 -20368.507,E2 -20368.507} C_VEL
LIN {X 0,Y 220.788,Z 278.482,A -85,B 0,C 180,E1 -20372.746,E2 -20372.746} C_VEL
LIN {X 0,Y 220.806,Z 278.48,A -85,B 0,C 180,E1 -20377.278,E2 -20377.278} C_VEL
LIN {X 0,Y 220.824,Z 278.48,A -85,B 0,C 180,E1 -20381.923,E2 -20381.923} C_VEL
LIN {X 0,Y 220.831,Z 278.476,A -85,B 0,C 180,E1 -20385.562,E2 -20385.562} C_VEL
LIN {X 0,Y 220.815,Z 278.48,A -85,B 0,C 180,E1 -20390.466,E2 -20390.466} C_VEL
LIN {X 0,Y 220.771,Z 278.485,A -85,B 0,C 180,E1 -20395.041,E2 -20395.041} C_VEL
LIN {X 0,Y 220.803,Z 278.615,A -85,B 0,C 180,E1 -20395.723,E2 -20395.723} C_VEL
LIN {X 0,Y 221.895,Z 281.476,A -85,B 0,C 180,E1 -20396.064,E2 -20396.064} C_VEL
LIN {X 0,Y 223.205,Z 283.615,A -85,B 0,C 180,E1 -20396.4,E2 -20396.4} C_VEL
LIN {X 0,Y 228.191,Z 293.201,A -85,B 0,C 180,E1 -20397.858,E2 -20397.858} C_VEL
LIN {X 0,Y 232.611,Z 302.984,A -85,B 0,C 180,E1 -20399.411,E2 -20399.411} C_VEL
LIN {X 0,Y 236.633,Z 313.857,A -85,B 0,C 180,E1 -20401.226,E2 -20401.226} C_VEL
LIN {X 0,Y 240.262,Z 322.88,A -85,B 0,C 180,E1 -20402.971,E2 -20402.971} C_VEL
LIN {X 0,Y 244.554,Z 331.01,A -85,B 0,C 180,E1 -20404.825,E2 -20404.825} C_VEL
LIN {X 0,Y 251.165,Z 340.733,A -85,B 0,C 180,E1 -20407.394,E2 -20407.394} C_VEL
LIN {X 0,Y 259.4,Z 350.084,A -85,B 0,C 180,E1 -20410.266,E2 -20410.266} C_VEL
LIN {X 0,Y 268.661,Z 358.706,A -85,B 0,C 180,E1 -20413.277,E2 -20413.277} C_VEL
LIN {X 0,Y 275.79,Z 364.375,A -85,B 0,C 180,E1 -20415.501,E2 -20415.501} C_VEL
LIN {X 0,Y 283.145,Z 369.915,A -85,B 0,C 180,E1 -20417.912,E2 -20417.912} C_VEL
LIN {X 0,Y 289.608,Z 374.527,A -85,B 0,C 180,E1 -20420.22,E2 -20420.22} C_VEL
LIN {X 0,Y 295.208,Z 378.273,A -85,B 0,C 180,E1 -20422.476,E2 -20422.476} C_VEL
LIN {X 0,Y 297.046,Z 379.67,A -85,B 0,C 180,E1 -20423.466,E2 -20423.466} C_VEL
LIN {X 0,Y 300.809,Z 382.386,A -85,B 0,C 180,E1 -20425.981,E2 -20425.981} C_VEL
LIN {X 0,Y 302.651,Z 383.327,A -85,B 0,C 180,E1 -20427.338,E2 -20427.338} C_VEL
LIN {X 0,Y 304.005,Z 383.887,A -85,B 0,C 180,E1 -20428.675,E2 -20428.675} C_VEL
LIN {X 0,Y 304.753,Z 384.071,A -85,B 0,C 180,E1 -20430,E2 -20430} C_VEL
LIN {X 0,Y 303.986,Z 383.888,A -85,B 0,C 180,E1 -20431.325,E2 -20431.325} C_VEL
LIN {X 0,Y 302.495,Z 383.267,A -85,B 0,C 180,E1 -20432.761,E2 -20432.761} C_VEL
LIN {X 0,Y 300.793,Z 382.386,A -85,B 0,C 180,E1 -20434.019,E2 -20434.019} C_VEL
LIN {X 0,Y 297.046,Z 379.669,A -85,B 0,C 180,E1 -20436.534,E2 -20436.534} C_VEL
LIN {X 0,Y 295.191,Z 378.273,A -85,B 0,C 180,E1 -20437.524,E2 -20437.524} C_VEL
LIN {X 0,Y 289.647,Z 374.526,A -85,B 0,C 180,E1 -20439.779,E2 -20439.779} C_VEL
LIN {X 0,Y 285.333,Z 371.438,A -85,B 0,C 180,E1 -20441.364,E2 -20441.364} C_VEL
LIN {X 0,Y 278.075,Z 366.137,A -85,B 0,C 180,E1 -20443.767,E2 -20443.767} C_VEL
LIN {X 0,Y 270.608,Z 360.325,A -85,B 0,C 180,E1 -20446.112,E2 -20446.112} C_VEL
LIN {X 0,Y 262.408,Z 353.023,A -85,B 0,C 180,E1 -20448.747,E2 -20448.747} C_VEL
LIN {X 0,Y 254.847,Z 345.145,A -85,B 0,C 180,E1 -20451.291,E2 -20451.291} C_VEL
LIN {X 0,Y 248.801,Z 337.626,A -85,B 0,C 180,E1 -20453.47,E2 -20453.47} C_VEL
LIN {X 0,Y 243.366,Z 328.936,A -85,B 0,C 180,E1 -20455.668,E2 -20455.668} C_VEL
LIN {X 0,Y 239.035,Z 320.169,A -85,B 0,C 180,E1 -20457.585,E2 -20457.585} C_VEL
LIN {X 0,Y 235.358,Z 310.287,A -85,B 0,C 180,E1 -20459.389,E2 -20459.389} C_VEL
LIN {X 0,Y 231.283,Z 299.809,A -85,B 0,C 180,E1 -20461.102,E2 -20461.102} C_VEL
LIN {X 0,Y 225.51,Z 287.884,A -85,B 0,C 180,E1 -20462.976,E2 -20462.976} C_VEL
LIN {X 0,Y 222.322,Z 282.062,A -85,B 0,C 180,E1 -20463.852,E2 -20463.852} C_VEL
LIN {X 0,Y 220.932,Z 279.314,A -85,B 0,C 180,E1 -20464.224,E2 -20464.224} C_VEL
LIN {X 0,Y 220.779,Z 278.485,A -85,B 0,C 180,E1 -20464.353,E2 -20464.353} C_VEL
LIN {X 0,Y 220.796,Z 278.482,A -85,B 0,C 180,E1 -20467.295,E2 -20467.295} C_VEL
LIN {X 0,Y 220.819,Z 278.48,A -85,B 0,C 180,E1 -20471.94,E2 -20471.94} C_VEL
LIN {X 0,Y 220.831,Z 278.477,A -85,B 0,C 180,E1 -20475.579,E2 -20475.579} C_VEL
LIN {X 0,Y 220.822,Z 278.478,A -85,B 0,C 180,E1 -20480.483,E2 -20480.483} C_VEL
LIN {X 0,Y 220.783,Z 278.483,A -85,B 0,C 180,E1 -20485.057,E2 -20485.057} C_VEL
LIN {X 0,Y 220.806,Z 278.48,A -85,B 0,C 180,E1 -20489.4,E2 -20489.4} C_VEL
LIN {X 0,Y 220.866,Z 278.471,A -85,B 0,C 180,E1 -20493.559,E2 -20493.559} C_VEL
LIN {X 0,Y 220.832,Z 278.478,A -85,B 0,C 180,E1 -20497.561,E2 -20497.561} C_VEL
LIN {X 0,Y 220.902,Z 278.468,A -85,B 0,C 180,E1 -20502.636,E2 -20502.636} C_VEL
LIN {X 0,Y 220.976,Z 278.46,A -85,B 0,C 180,E1 -20507.148,E2 -20507.148} C_VEL
LIN {X 0,Y 221.184,Z 278.428,A -85,B 0,C 180,E1 -20510.87,E2 -20510.87} C_VEL
LIN {X 0,Y 221.117,Z 278.44,A -85,B 0,C 180,E1 -20514.539,E2 -20514.539} C_VEL
LIN {X 0,Y 221.501,Z 278.367,A -85,B 0,C 180,E1 -20518.192,E2 -20518.192} C_VEL
LIN {X 0,Y 221.466,Z 278.394,A -85,B 0,C 180,E1 -20521.829,E2 -20521.829} C_VEL
LIN {X 0,Y 221.244,Z 278.426,A -85,B 0,C 180,E1 -20527.31,E2 -20527.31} C_VEL
LIN {X 0,Y 221.063,Z 278.45,A -85,B 0,C 180,E1 -20531.007,E2 -20531.007} C_VEL
LIN {X 0,Y 220.981,Z 278.461,A -85,B 0,C 180,E1 -20536.643,E2 -20536.643} C_VEL
LIN {X 0,Y 220.859,Z 278.475,A -85,B 0,C 180,E1 -20540.499,E2 -20540.499} C_VEL
LIN {X 0,Y 220.817,Z 278.481,A -85,B 0,C 180,E1 -20544.451,E2 -20544.451} C_VEL
LIN {X 0,Y 220.863,Z 278.475,A -85,B 0,C 180,E1 -20547.006,E2 -20547.006} C_VEL
LIN {X 0,Y 220.995,Z 279.732,A -85,B 0,C 180,E1 -20550.838,E2 -20550.838} C_VEL
LIN {X 0,Y 221.206,Z 281.497,A -85,B 0,C 180,E1 -20554.892,E2 -20554.892} C_VEL
LIN {X 0,Y 221.551,Z 283.661,A -85,B 0,C 180,E1 -20559.389,E2 -20559.389} C_VEL
LIN {X 0,Y 221.769,Z 285.702,A -85,B 0,C 180,E1 -20563.209,E2 -20563.209} C_VEL
LIN {X 0,Y 221.731,Z 287.776,A -85,B 0,C 180,E1 -20566.815,E2 -20566.815} C_VEL
LIN {X 0,Y 221.358,Z 290.145,A -85,B 0,C 180,E1 -20570.582,E2 -20570.582} C_VEL
LIN {X 0,Y 221.047,Z 291.632,A -85,B 0,C 180,E1 -20572.838,E2 -20572.838} C_VEL
LIN {X 0,Y 220.534,Z 293.739,A -85,B 0,C 180,E1 -20575.914,E2 -20575.914} C_VEL
LIN {X 0,Y 221.468,Z 297.097,A -85,B 0,C 180,E1 -20576.276,E2 -20576.276} C_VEL
LIN {X 0,Y 225.285,Z 309.217,A -85,B 0,C 180,E1 -20577.855,E2 -20577.855} C_VEL
LIN {X 0,Y 227.787,Z 319.637,A -85,B 0,C 180,E1 -20579.335,E2 -20579.335} C_VEL
LIN {X 0,Y 229.474,Z 329.923,A -85,B 0,C 180,E1 -20580.935,E2 -20580.935} C_VEL
LIN {X 0,Y 230.357,Z 339.151,A -85,B 0,C 180,E1 -20582.526,E2 -20582.526} C_VEL
LIN {X 0,Y 230.575,Z 348.133,A -85,B 0,C 180,E1 -20584.257,E2 -20584.257} C_VEL
LIN {X 0,Y 230.343,Z 351.554,A -85,B 0,C 180,E1 -20584.955,E2 -20584.955} C_VEL
LIN {X 0,Y 227.486,Z 362.266,A -85,B 0,C 180,E1 -20587.284,E2 -20587.284} C_VEL
LIN {X 0,Y 227.281,Z 363.007,A -85,B 0,C 180,E1 -20587.481,E2 -20587.481} C_VEL
LIN {X 0,Y 225.591,Z 367.091,A -85,B 0,C 180,E1 -20588.507,E2 -20588.507} C_VEL
LIN {X 0,Y 221.196,Z 373.121,A -85,B 0,C 180,E1 -20590.158,E2 -20590.158} C_VEL
LIN {X 0,Y 216.829,Z 378.652,A -85,B 0,C 180,E1 -20591.982,E2 -20591.982} C_VEL
LIN {X 0,Y 215.21,Z 381.639,A -85,B 0,C 180,E1 -20593.264,E2 -20593.264} C_VEL
LIN {X 0,Y 213.713,Z 386.432,A -85,B 0,C 180,E1 -20595.722,E2 -20595.722} C_VEL
LIN {X 0,Y 212.589,Z 390.761,A -85,B 0,C 180,E1 -20598.56,E2 -20598.56} C_VEL
LIN {X 0,Y 212.081,Z 393.132,A -85,B 0,C 180,E1 -20600.463,E2 -20600.463} C_VEL
LIN {X 0,Y 211.674,Z 394.934,A -85,B 0,C 180,E1 -20602.368,E2 -20602.368} C_VEL
LIN {X 0,Y 211.379,Z 397.388,A -85,B 0,C 180,E1 -20606.187,E2 -20606.187} C_VEL
LIN {X 0,Y 211.434,Z 397.983,A -85,B 0,C 180,E1 -20608.095,E2 -20608.095} C_VEL
LIN {X 0,Y 211.526,Z 398.141,A -85,B 0,C 180,E1 -20610,E2 -20610} C_VEL
LIN {X 0,Y 211.434,Z 397.983,A -85,B 0,C 180,E1 -20611.905,E2 -20611.905} C_VEL
LIN {X 0,Y 211.395,Z 397.312,A -85,B 0,C 180,E1 -20614.048,E2 -20614.048} C_VEL
LIN {X 0,Y 211.668,Z 394.934,A -85,B 0,C 180,E1 -20617.632,E2 -20617.632} C_VEL
LIN {X 0,Y 212.32,Z 391.98,A -85,B 0,C 180,E1 -20620.489,E2 -20620.489} C_VEL
LIN {X 0,Y 213.261,Z 387.986,A -85,B 0,C 180,E1 -20623.337,E2 -20623.337} C_VEL
LIN {X 0,Y 214.799,Z 382.856,A -85,B 0,C 180,E1 -20626.147,E2 -20626.147} C_VEL
LIN {X 0,Y 216.377,Z 377.593,A -85,B 0,C 180,E1 -20628.462,E2 -20628.462} C_VEL
LIN {X 0,Y 218.38,Z 371.28,A -85,B 0,C 180,E1 -20630.732,E2 -20630.732} C_VEL
LIN {X 0,Y 219.965,Z 365.324,A -85,B 0,C 180,E1 -20632.544,E2 -20632.544} C_VEL
LIN {X 0,Y 221.916,Z 358.399,A -85,B 0,C 180,E1 -20634.311,E2 -20634.311} C_VEL
LIN {X 0,Y 223.815,Z 351.356,A -85,B 0,C 180,E1 -20635.828,E2 -20635.828} C_VEL
LIN {X 0,Y 223.836,Z 341.788,A -85,B 0,C 180,E1 -20637.814,E2 -20637.814} C_VEL
LIN {X 0,Y 223.316,Z 334.648,A -85,B 0,C 180,E1 -20639.171,E2 -20639.171} C_VEL
LIN {X 0,Y 222.009,Z 324.677,A -85,B 0,C 180,E1 -20640.87,E2 -20640.87} C_VEL
LIN {X 0,Y 219.828,Z 314.15,A -85,B 0,C 180,E1 -20642.506,E2 -20642.506} C_VEL
LIN {X 0,Y 216.898,Z 303.777,A -85,B 0,C 180,E1 -20644.001,E2 -20644.001} C_VEL
LIN {X 0,Y 214.375,Z 296.55,A -85,B 0,C 180,E1 -20645.017,E2 -20645.017} C_VEL
LIN {X 0,Y 213.617,Z 293.623,A -85,B 0,C 180,E1 -20645.322,E2 -20645.322} C_VEL
LIN {X 0,Y 214.134,Z 291.437,A -85,B 0,C 180,E1 -20648.578,E2 -20648.578} C_VEL
LIN {X 0,Y 214.49,Z 289.861,A -85,B 0,C 180,E1 -20651.082,E2 -20651.082} C_VEL
LIN {X 0,Y 214.704,Z 288.178,A -85,B 0,C 180,E1 -20653.922,E2 -20653.922} C_VEL
LIN {X 0,Y 214.74,Z 286.686,A -85,B 0,C 180,E1 -20656.573,E2 -20656.573} C_VEL
LIN {X 0,Y 214.636,Z 285.37,A -85,B 0,C 180,E1 -20659.078,E2 -20659.078} C_VEL
LIN {X 0,Y 214.25,Z 283.104,A -85,B 0,C 180,E1 -20663.8,E2 -20663.8} C_VEL
LIN {X 0,Y 213.995,Z 281.019,A -85,B 0,C 180,E1 -20668.635,E2 -20668.635} C_VEL
LIN {X 0,Y 213.803,Z 279.515,A -85,B 0,C 180,E1 -20672.59,E2 -20672.59} C_VEL
LIN {X 0,Y 213.804,Z 279.355,A -85,B 0,C 180,E1 -20676.98,E2 -20676.98} C_VEL
LIN {X 0,Y 213.891,Z 279.342,A -85,B 0,C 180,E1 -20682.789,E2 -20682.789} C_VEL
LIN {X 0,Y 213.935,Z 279.336,A -85,B 0,C 180,E1 -20686.695,E2 -20686.695} C_VEL
LIN {X 0,Y 214.136,Z 279.31,A -85,B 0,C 180,E1 -20690.544,E2 -20690.544} C_VEL
LIN {X 0,Y 214.078,Z 279.317,A -85,B 0,C 180,E1 -20694.337,E2 -20694.337} C_VEL
LIN {X 0,Y 214.403,Z 279.274,A -85,B 0,C 180,E1 -20698.111,E2 -20698.111} C_VEL
LIN {X 0,Y 214.534,Z 279.246,A -85,B 0,C 180,E1 -20699.989,E2 -20699.989} C_VEL
LIN {X 0,Y 214.434,Z 279.246,A -85,B 0,C 180,E1 -20701.867,E2 -20701.867} C_VEL
LIN {X 0,Y 214.176,Z 279.305,A -85,B 0,C 180,E1 -20707.531,E2 -20707.531} C_VEL
LIN {X 0,Y 213.978,Z 279.331,A -85,B 0,C 180,E1 -20711.354,E2 -20711.354} C_VEL
LIN {X 0,Y 213.879,Z 279.339,A -85,B 0,C 180,E1 -20715.228,E2 -20715.228} C_VEL
LIN {X 0,Y 213.775,Z 279.35,A -85,B 0,C 180,E1 -20719.18,E2 -20719.18} C_VEL
LIN {X 0,Y 213.774,Z 279.354,A -85,B 0,C 180,E1 -20723.222,E2 -20723.222} C_VEL
LIN {X 0,Y 213.786,Z 279.354,A -85,B 0,C 180,E1 -20727.43,E2 -20727.43} C_VEL
LIN {X 0,Y 213.732,Z 279.361,A -85,B 0,C 180,E1 -20731.728,E2 -20731.728} C_VEL
LIN {X 0,Y 213.721,Z 279.363,A -85,B 0,C 180,E1 -20736.276,E2 -20736.276} C_VEL
LIN {X 0,Y 213.761,Z 279.357,A -85,B 0,C 180,E1 -20741.096,E2 -20741.096} C_VEL
LIN {X 0,Y 213.8,Z 279.353,A -85,B 0,C 180,E1 -20743.684,E2 -20743.684} C_VEL
LIN {X 0,Y 213.773,Z 279.357,A -85,B 0,C 180,E1 -20746.34,E2 -20746.34} C_VEL
LIN {X 0,Y 213.756,Z 279.358,A -85,B 0,C 180,E1 -20749.11,E2 -20749.11} C_VEL
LIN {X 0,Y 213.71,Z 279.366,A -85,B 0,C 180,E1 -20753.706,E2 -20753.706} C_VEL
LIN {X 0,Y 213.724,Z 279.367,A -85,B 0,C 180,E1 -20754.448,E2 -20754.448} C_VEL
LIN {X 0,Y 214.7,Z 282.165,A -85,B 0,C 180,E1 -20754.787,E2 -20754.787} C_VEL
LIN {X 0,Y 216.122,Z 284.309,A -85,B 0,C 180,E1 -20755.168,E2 -20755.168} C_VEL
LIN {X 0,Y 221.267,Z 294.052,A -85,B 0,C 180,E1 -20756.774,E2 -20756.774} C_VEL
LIN {X 0,Y 226.251,Z 305.06,A -85,B 0,C 180,E1 -20758.649,E2 -20758.649} C_VEL
